KUKA KRL program: MyProgram_217().src

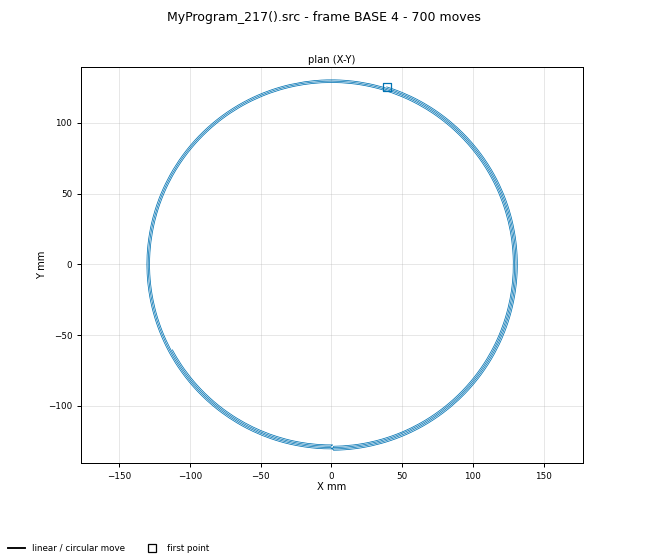
[picture p0: tool path of MyProgram_217().src in frame BASE 4, 700 of 700 moves have a stored position in this frame; points joined in program order, loops and branches not executed]
&ACCESS RVP
&REL 1
&PARAM TEMPLATE = C:\KRC\Roboter\Template\vorgabe
&PARAM EDITMASK = *
DEF MyProgram_217()
; ---- Setting reference (Base) ----
$BASE = BASE_DATA[4]

; --------------------------
; ---- Setting tool (TCP) ----
$TOOL = TOOL_DATA[3]
; --------------------------

$VEL.CP = VEL_APROX_PRINT
Startdeposition()
$VEL.CP = VEL_PRINT
LIN {X 39.0759,Y 125.4195,Z 152,A 69.1169,B 22.3843,C -1.1752,E1 22.4627,E2 378.1488} C_DIS
LIN {X 42.8509,Y 124.1788,Z 152,A 67.5035,B 22.3841,C -1.1792,E1 22.4669,E2 379.7481} C_DIS
LIN {X 46.0202,Y 123.0393,Z 152,A 66.1217,B 22.384,C -1.1819,E1 22.4705,E2 381.1197} C_DIS
LIN {X 49.9531,Y 121.4979,Z 152,A 64.0828,B 22.3845,C -1.1709,E1 22.4758,E2 383.1823} C_DIS
LIN {X 53.3923,Y 120.0244,Z 152,A 62.6413,B 22.3842,C -1.1779,E1 22.4795,E2 384.6014} C_DIS
LIN {X 55.8372,Y 118.9089,Z 152,A 61.2764,B 22.3847,C -1.1675,E1 22.483,E2 385.9896} C_DIS
LIN {X 59.0575,Y 117.3417,Z 152,A 59.7473,B 22.3847,C -1.167,E1 22.4868,E2 387.5152} C_DIS
LIN {X 62.6882,Y 115.4438,Z 152,A 57.9615,B 22.3848,C -1.1646,E1 22.4912,E2 389.3015} C_DIS
LIN {X 65.3716,Y 113.9459,Z 152,A 56.5252,B 22.3851,C -1.1582,E1 22.4947,E2 390.7497} C_DIS
LIN {X 69.7331,Y 111.3304,Z 152,A 54.6879,B 22.3844,C -1.1727,E1 22.499,E2 392.5428} C_DIS
LIN {X 72.7495,Y 109.3827,Z 152,A 52.8465,B 22.3852,C -1.1572,E1 22.5034,E2 394.4178} C_DIS
LIN {X 76.5216,Y 106.7777,Z 152,A 50.8731,B 22.3852,C -1.155,E1 22.5079,E2 396.3891} C_DIS
LIN {X 80.0679,Y 104.1454,Z 152,A 48.9647,B 22.3854,C -1.1524,E1 22.5121,E2 398.2966} C_DIS
LIN {X 83.4471,Y 101.4582,Z 152,A 47.0498,B 22.3857,C -1.1473,E1 22.5163,E2 400.2166} C_DIS
LIN {X 86.8041,Y 98.6009,Z 152,A 45.3735,B 22.3853,C -1.1552,E1 22.5198,E2 401.8648} C_DIS
LIN {X 88.621,Y 96.9709,Z 152,A 44.0641,B 22.3859,C -1.1415,E1 22.5226,E2 403.2042} C_DIS
LIN {X 92.4956,Y 93.2824,Z 152,A 41.7817,B 22.3861,C -1.1389,E1 22.5271,E2 405.4825} C_DIS
LIN {X 95.519,Y 90.1839,Z 152,A 39.8997,B 22.3862,C -1.1351,E1 22.5308,E2 407.3654} C_DIS
LIN {X 98.6375,Y 86.7627,Z 152,A 37.8778,B 22.3865,C -1.1304,E1 22.5346,E2 409.3894} C_DIS
LIN {X 101.415,Y 83.4994,Z 152,A 36.2489,B 22.3861,C -1.1374,E1 22.5374,E2 410.9914} C_DIS
LIN {X 103.0184,Y 81.5129,Z 152,A 34.8749,B 22.3869,C -1.1223,E1 22.5399,E2 412.3977} C_DIS
LIN {X 105.772,Y 77.9059,Z 152,A 32.9472,B 22.3869,C -1.1199,E1 22.5431,E2 414.3213} C_DIS
LIN {X 107.9986,Y 74.7891,Z 152,A 31.2247,B 22.3873,C -1.1132,E1 22.5459,E2 416.0518} C_DIS
LIN {X 110.566,Y 70.9379,Z 152,A 29.2946,B 22.3873,C -1.1122,E1 22.5488,E2 417.9735} C_DIS
LIN {X 112.9802,Y 67.0265,Z 152,A 27.2685,B 22.3876,C -1.1058,E1 22.5518,E2 420.0046} C_DIS
LIN {X 115.1352,Y 63.254,Z 152,A 25.4004,B 22.3878,C -1.102,E1 22.5543,E2 421.8718} C_DIS
LIN {X 116.9711,Y 59.7855,Z 152,A 23.8677,B 22.3876,C -1.1059,E1 22.5563,E2 423.385} C_DIS
LIN {X 118.8063,Y 56.0533,Z 152,A 21.862,B 22.3883,C -1.0915,E1 22.5587,E2 425.4161} C_DIS
LIN {X 120.4751,Y 52.3674,Z 152,A 20.2435,B 22.3883,C -1.0935,E1 22.5605,E2 427.0193} C_DIS
LIN {X 121.5852,Y 49.7396,Z 152,A 19.0427,B 22.3883,C -1.092,E1 22.5618,E2 428.2167} C_DIS
LIN {X 123.0594,Y 45.9666,Z 152,A 17.2165,B 22.3887,C -1.084,E1 22.5637,E2 430.0524} C_DIS
LIN {X 124.4991,Y 41.9132,Z 152,A 15.3852,B 22.3888,C -1.0805,E1 22.5653,E2 431.881} C_DIS
LIN {X 125.5845,Y 38.537,Z 152,A 13.7778,B 22.3892,C -1.0729,E1 22.5667,E2 433.4979} C_DIS
LIN {X 126.8539,Y 34.1282,Z 152,A 11.8493,B 22.3892,C -1.0704,E1 22.5681,E2 435.4206} C_DIS
LIN {X 127.5693,Y 31.3524,Z 152,A 10.4272,B 22.3898,C -1.0581,E1 22.5691,E2 436.8654} C_DIS
LIN {X 128.3238,Y 28.1021,Z 152,A 8.5123,B 22.391,C -1.0313,E1 22.5703,E2 438.8375} C_DIS
LIN {X 129.3311,Y 23.0236,Z 152,A 6.9093,B 22.3899,C -1.056,E1 22.5711,E2 440.3655} C_DIS
LIN {X 129.9659,Y 19.125,Z 152,A 5.1562,B 22.3902,C -1.0491,E1 22.5718,E2 442.1251} C_DIS
LIN {X 130.4075,Y 15.8299,Z 152,A 3.6744,B 22.3905,C -1.043,E1 22.5723,E2 443.613} C_DIS
LIN {X 130.9161,Y 10.8465,Z 152,A 1.5967,B 22.3905,C -1.0412,E1 22.5729,E2 445.6813} C_DIS
LIN {X 131.1931,Y 6.7104,Z 152,A -0.1239,B 22.3906,C -1.0397,E1 22.5732,E2 447.3943} C_DIS
LIN {X 131.3377,Y 2.7109,Z 152,A -1.9941,B 22.3912,C -1.028,E1 22.5733,E2 449.2825} C_DIS
LIN {X 131.3529,Y -1.7959,Z 152,A -3.9022,B 22.3913,C -1.0245,E1 22.5733,E2 451.187} C_DIS
LIN {X 131.2356,Y -5.864,Z 152,A -5.7352,B 22.3917,C -1.0159,E1 22.5731,E2 453.0299} C_DIS
LIN {X 131.0106,Y -9.6365,Z 152,A -7.2728,B 22.3917,C -1.0161,E1 22.5728,E2 454.5569} C_DIS
LIN {X 130.6589,Y -13.604,Z 152,A -9.1407,B 22.3922,C -1.004,E1 22.5723,E2 456.4436} C_DIS
LIN {X 130.0858,Y -18.286,Z 152,A -11.0585,B 22.3922,C -1.0043,E1 22.5716,E2 458.348} C_DIS
LIN {X 129.5248,Y -21.9092,Z 152,A -12.6685,B 22.3924,C -0.9986,E1 22.5709,E2 459.9622} C_DIS
LIN {X 128.7591,Y -26.0326,Z 152,A -14.5575,B 22.3928,C -0.9898,E1 22.5699,E2 461.8616} C_DIS
LIN {X 127.7964,Y -30.4103,Z 152,A -16.4042,B 22.3928,C -0.9889,E1 22.5687,E2 463.6986} C_DIS
LIN {X 126.9735,Y -33.6799,Z 152,A -17.7135,B 22.3927,C -0.9921,E1 22.5678,E2 464.9909} C_DIS
LIN {X 126.1061,Y -36.7942,Z 152,A -19.2732,B 22.3932,C -0.9804,E1 22.5666,E2 466.5712} C_DIS
LIN {X 124.8598,Y -40.8297,Z 152,A -21.1531,B 22.3935,C -0.9727,E1 22.565,E2 468.459} C_DIS
LIN {X 123.6518,Y -44.3489,Z 152,A -22.6966,B 22.3935,C -0.9716,E1 22.5636,E2 469.9957} C_DIS
LIN {X 122.4904,Y -47.462,Z 152,A -24.0809,B 22.3935,C -0.9703,E1 22.5622,E2 471.3746} C_DIS
LIN {X 120.3805,Y -52.5861,Z 152,A -26.6321,B 22.3942,C -0.9564,E1 22.5595,E2 473.9463} C_DIS
LIN {X 118.6274,Y -56.4278,Z 152,A -28.3416,B 22.3942,C -0.9573,E1 22.5575,E2 475.6429} C_DIS
LIN {X 115.2676,Y -63.0113,Z 152,A -31.5961,B 22.3946,C -0.9462,E1 22.5533,E2 478.9068} C_DIS
LIN {X 113.0629,Y -66.8877,Z 152,A -33.5919,B 22.3949,C -0.9381,E1 22.5504,E2 480.9122} C_DIS
LIN {X 110.7037,Y -70.7228,Z 152,A -35.4887,B 22.3949,C -0.9358,E1 22.5476,E2 482.8041} C_DIS
LIN {X 108.293,Y -74.3616,Z 152,A -37.3931,B 22.3952,C -0.9305,E1 22.5447,E2 484.7118} C_DIS
LIN {X 105.6688,Y -78.0464,Z 152,A -39.3055,B 22.3952,C -0.9281,E1 22.5415,E2 486.6201} C_DIS
LIN {X 103.8884,Y -80.4004,Z 152,A -40.7022,B 22.3956,C -0.9193,E1 22.5391,E2 488.0322} C_DIS
LIN {X 101.1979,Y -83.7616,Z 152,A -43.1794,B 22.3969,C -0.8855,E1 22.5346,E2 490.5846} C_DIS
LIN {X 97.4652,Y -88.0773,Z 152,A -45.38,B 22.3966,C -0.893,E1 22.5306,E2 492.7545} C_DIS
LIN {X 94.5654,Y -91.183,Z 152,A -46.9074,B 22.3962,C -0.9041,E1 22.5277,E2 494.2455} C_DIS
LIN {X 89.8695,Y -95.8156,Z 152,A -49.6238,B 22.3962,C -0.905,E1 22.5223,E2 496.9468} C_DIS
LIN {X 84.2334,Y -100.8059,Z 152,A -52.7429,B 22.3962,C -0.9054,E1 22.5158,E2 500.0509} C_DIS
LIN {X 82.4164,Y -102.2964,Z 152,A -54.3606,B 22.3973,C -0.8747,E1 22.5121,E2 501.7419} C_DIS
LIN {X 79.0783,Y -104.8983,Z 152,A -56.1035,B 22.3973,C -0.8758,E1 22.5082,E2 503.475} C_DIS
LIN {X 76.025,Y -107.1324,Z 152,A -57.4826,B 22.3969,C -0.8853,E1 22.5051,E2 504.8237} C_DIS
LIN {X 72.219,Y -109.7335,Z 152,A -59.4323,B 22.3969,C -0.8843,E1 22.5006,E2 506.7687} C_DIS
LIN {X 68.385,Y -112.1635,Z 152,A -61.4412,B 22.3972,C -0.8792,E1 22.4958,E2 508.7837} C_DIS
LIN {X 64.5104,Y -114.4354,Z 152,A -63.3541,B 22.3972,C -0.8779,E1 22.4912,E2 510.6936} C_DIS
LIN {X 60.7291,Y -116.4844,Z 152,A -65.095,B 22.3971,C -0.8811,E1 22.487,E2 512.4203} C_DIS
LIN {X 56.5099,Y -118.5882,Z 152,A -67.198,B 22.3973,C -0.8756,E1 22.4817,E2 514.5314} C_DIS
LIN {X 53.0564,Y -120.1746,Z 152,A -68.9498,B 22.3976,C -0.8686,E1 22.4772,E2 516.2966} C_DIS
LIN {X 49.5085,Y -121.6783,Z 152,A -70.4769,B 22.3974,C -0.8735,E1 22.4733,E2 517.807} C_DIS
LIN {X 45.1537,Y -123.3616,Z 152,A -72.6362,B 22.3977,C -0.8649,E1 22.4676,E2 519.9834} C_DIS
LIN {X 41.6015,Y -124.6029,Z 152,A -74.081,B 22.3974,C -0.8722,E1 22.4639,E2 521.406} C_DIS
LIN {X 38.537,Y -125.5845,Z 152,A -75.5338,B 22.3976,C -0.8682,E1 22.46,E2 522.8662} C_DIS
LIN {X 35.354,Y -126.5174,Z 152,A -76.8689,B 22.3974,C -0.8719,E1 22.4564,E2 524.1891} C_DIS
LIN {X 31.0295,Y -127.6472,Z 152,A -78.8275,B 22.3975,C -0.8694,E1 22.4511,E2 526.1506} C_DIS
LIN {X 28.7199,Y -128.1875,Z 152,A -80.4521,B 22.3986,C -0.841,E1 22.4465,E2 527.8474} C_DIS
LIN {X 24.8562,Y -128.9914,Z 152,A -82.107,B 22.3985,C -0.8426,E1 22.442,E2 529.4957} C_DIS
LIN {X 21.1843,Y -129.6457,Z 152,A -83.4884,B 22.3981,C -0.8528,E1 22.4382,E2 530.8489} C_DIS
LIN {X 16.9785,Y -130.2626,Z 152,A -85.2127,B 22.398,C -0.8576,E1 22.4335,E2 532.5589} C_DIS
LIN {X 12.8893,Y -130.731,Z 152,A -87.043,B 22.398,C -0.855,E1 22.4284,E2 534.3946} C_DIS
LIN {X 9.8072,Y -130.9981,Z 152,A -88.5323,B 22.3983,C -0.8479,E1 22.4242,E2 535.9016} C_DIS
LIN {X 5.3117,Y -131.2573,Z 152,A -90.3189,B 22.398,C -0.8553,E1 22.4193,E2 537.668} C_DIS
LIN {X 1.4511,Y -131.3586,Z 152,A -92.1085,B 22.3982,C -0.85,E1 22.4143,E2 539.4713} C_DIS
LIN {X 1.4511,Y -131.3586,Z 152,A -92.1085,B 22.3982,C -0.85,E1 22.4143,E2 539.4713} C_DIS
Enddeposition()
LIN {X 0.9252,Y -130.4174,Z 152,A -91.4009,B 21.3974,C -0.7347,E1 21.4116,E2 538.9603} C_DIS
Startdeposition()
$VEL.CP = VEL_PRINT
LIN {X 4.401,Y -130.3502,Z 152,A -89.5833,B 21.397,C -0.7479,E1 21.4168,E2 537.1069} C_DIS
LIN {X 7.5621,Y -130.2041,Z 152,A -87.7196,B 21.3963,C -0.7696,E1 21.4221,E2 535.1847} C_DIS
LIN {X 12.3533,Y -129.8363,Z 152,A -86.2062,B 21.3971,C -0.7439,E1 21.4261,E2 533.7428} C_DIS
LIN {X 16.3199,Y -129.399,Z 152,A -84.4088,B 21.3971,C -0.7469,E1 21.4311,E2 531.9389} C_DIS
LIN {X 22.9385,Y -128.3895,Z 152,A -81.4914,B 21.3971,C -0.7479,E1 21.4392,E2 529.0222} C_DIS
LIN {X 29.5447,Y -127.033,Z 152,A -78.4786,B 21.3968,C -0.7527,E1 21.4474,E2 526.0009} C_DIS
LIN {X 34.0528,Y -125.8993,Z 152,A -76.4296,B 21.3968,C -0.755,E1 21.453,E2 523.9493} C_DIS
LIN {X 38.0089,Y -124.7611,Z 152,A -74.7239,B 21.3968,C -0.7524,E1 21.4575,E2 522.2544} C_DIS
LIN {X 41.3367,Y -123.6984,Z 152,A -73.2639,B 21.3969,C -0.7508,E1 21.4614,E2 520.8018} C_DIS
LIN {X 44.246,Y -122.6877,Z 152,A -71.909,B 21.3969,C -0.7526,E1 21.4649,E2 519.4454} C_DIS
LIN {X 51.5801,Y -119.7894,Z 152,A -68.4066,B 21.3966,C -0.759,E1 21.474,E2 515.9348} C_DIS
LIN {X 54.631,Y -118.429,Z 152,A -66.0213,B 21.3951,C -0.8034,E1 21.4804,E2 513.4355} C_DIS
LIN {X 60.4214,Y -115.5822,Z 152,A -64.14,B 21.3965,C -0.7641,E1 21.4848,E2 511.6678} C_DIS
LIN {X 64.2221,Y -113.517,Z 152,A -62.1023,B 21.3961,C -0.7736,E1 21.4898,E2 509.6112} C_DIS
LIN {X 68.0638,Y -111.2555,Z 152,A -60.1772,B 21.3961,C -0.7757,E1 21.4944,E2 507.6876} C_DIS
LIN {X 71.6684,Y -108.9683,Z 152,A -58.3196,B 21.396,C -0.7784,E1 21.4987,E2 505.8297} C_DIS
LIN {X 75.4742,Y -106.3684,Z 152,A -56.4222,B 21.396,C -0.7766,E1 21.503,E2 503.9451} C_DIS
LIN {X 77.6887,Y -104.7616,Z 152,A -55.2144,B 21.396,C -0.7793,E1 21.5058,E2 502.735} C_DIS
LIN {X 82.2112,Y -101.2519,Z 152,A -52.5747,B 21.3955,C -0.7904,E1 21.5116,E2 500.0766} C_DIS
LIN {X 85.2765,Y -98.6834,Z 152,A -50.4735,B 21.3948,C -0.8103,E1 21.5161,E2 497.9308} C_DIS
LIN {X 88.3815,Y -95.9124,Z 152,A -48.5103,B 21.3945,C -0.8209,E1 21.5202,E2 495.9483} C_DIS
LIN {X 91.9267,Y -92.5199,Z 152,A -46.9023,B 21.3952,C -0.8004,E1 21.5233,E2 494.4042} C_DIS
LIN {X 97.2688,Y -86.8865,Z 152,A -43.0456,B 21.3941,C -0.8297,E1 21.5307,E2 490.4879} C_DIS
LIN {X 100.2547,Y -83.4239,Z 152,A -41.4961,B 21.3947,C -0.8133,E1 21.5334,E2 488.9914} C_DIS
LIN {X 102.7993,Y -80.2677,Z 152,A -39.7139,B 21.3946,C -0.818,E1 21.5365,E2 487.2063} C_DIS
LIN {X 105.4275,Y -76.7827,Z 152,A -37.8044,B 21.3944,C -0.8228,E1 21.5396,E2 485.2947} C_DIS
LIN {X 107.8695,Y -73.3123,Z 152,A -35.9707,B 21.3942,C -0.8265,E1 21.5426,E2 483.4617} C_DIS
LIN {X 110.366,Y -69.4969,Z 152,A -34.0103,B 21.3942,C -0.8301,E1 21.5455,E2 481.5032} C_DIS
LIN {X 112.6618,Y -65.711,Z 152,A -32.0287,B 21.3938,C -0.8373,E1 21.5483,E2 479.5141} C_DIS
LIN {X 114.6698,Y -62.1403,Z 152,A -29.1425,B 21.3917,C -0.8941,E1 21.5524,E2 476.4911} C_DIS
LIN {X 118.2409,Y -55.0378,Z 152,A -26.9035,B 21.3936,C -0.8448,E1 21.5549,E2 474.4006} C_DIS
LIN {X 121.0471,Y -48.5553,Z 152,A -23.7639,B 21.3931,C -0.8559,E1 21.5583,E2 471.2514} C_DIS
LIN {X 122.9923,Y -43.398,Z 152,A -21.3202,B 21.3928,C -0.8643,E1 21.5607,E2 468.801} C_DIS
LIN {X 124.1626,Y -39.921,Z 152,A -19.8445,B 21.3928,C -0.8629,E1 21.5619,E2 467.339} C_DIS
LIN {X 125.0716,Y -36.9756,Z 152,A -18.4548,B 21.3926,C -0.8688,E1 21.563,E2 465.9428} C_DIS
LIN {X 125.9647,Y -33.8073,Z 152,A -17.0128,B 21.3925,C -0.8731,E1 21.5641,E2 464.4988} C_DIS
LIN {X 126.9017,Y -30.1032,Z 152,A -15.3229,B 21.3923,C -0.8789,E1 21.5652,E2 462.8047} C_DIS
LIN {X 127.7436,Y -26.3,Z 152,A -13.6339,B 21.3921,C -0.8832,E1 21.5662,E2 461.1156} C_DIS
LIN {X 128.6323,Y -21.5356,Z 152,A -11.5618,B 21.3919,C -0.8873,E1 21.5672,E2 459.0468} C_DIS
LIN {X 129.1811,Y -17.9597,Z 152,A -10.0533,B 21.3919,C -0.8885,E1 21.5678,E2 457.5455} C_DIS
LIN {X 129.7907,Y -12.8285,Z 152,A -7.6059,B 21.3913,C -0.9041,E1 21.5686,E2 455.0729} C_DIS
LIN {X 130.1561,Y -8.3413,Z 152,A -5.7478,B 21.3913,C -0.9048,E1 21.569,E2 453.226} C_DIS
LIN {X 130.3399,Y -4.6658,Z 152,A -4.06,B 21.3909,C -0.9133,E1 21.5692,E2 451.527} C_DIS
LIN {X 130.4182,Y 1.2459,Z 152,A -1.5813,B 21.3908,C -0.916,E1 21.5692,E2 449.0586} C_DIS
LIN {X 130.2441,Y 6.8284,Z 152,A 0.9539,B 21.3903,C -0.9276,E1 21.569,E2 446.5096} C_DIS
LIN {X 129.9978,Y 10.5288,Z 152,A 2.8599,B 21.3895,C -0.9458,E1 21.5685,E2 444.5673} C_DIS
LIN {X 129.6462,Y 14.2119,Z 152,A 4.8108,B 21.3887,C -0.9664,E1 21.5679,E2 442.5741} C_DIS
LIN {X 128.9348,Y 19.646,Z 152,A 6.4917,B 21.3898,C -0.9396,E1 21.5673,E2 440.9781} C_DIS
LIN {X 128.1808,Y 24.0808,Z 152,A 8.89,B 21.3887,C -0.9656,E1 21.566,E2 438.5257} C_DIS
LIN {X 127.3556,Y 28.1238,Z 152,A 10.306,B 21.3893,C -0.9524,E1 21.5652,E2 437.1552} C_DIS
LIN {X 126.4429,Y 31.9722,Z 152,A 12.0043,B 21.3891,C -0.9559,E1 21.5641,E2 435.4592} C_DIS
LIN {X 125.3275,Y 36.1016,Z 152,A 13.8644,B 21.3889,C -0.9607,E1 21.5627,E2 433.5987} C_DIS
LIN {X 124.2876,Y 39.5299,Z 152,A 15.3719,B 21.3889,C -0.9623,E1 21.5614,E2 432.097} C_DIS
LIN {X 123.2775,Y 42.5754,Z 152,A 16.646,B 21.3889,C -0.9602,E1 21.5603,E2 430.8372} C_DIS
LIN {X 122.252,Y 45.4371,Z 152,A 17.902,B 21.3889,C -0.9604,E1 21.5591,E2 429.589} C_DIS
LIN {X 120.3818,Y 50.1816,Z 152,A 20.3347,B 21.3882,C -0.9758,E1 21.5566,E2 427.1303} C_DIS
LIN {X 119.1157,Y 53.117,Z 152,A 21.7307,B 21.3881,C -0.9794,E1 21.555,E2 425.7336} C_DIS
LIN {X 116.6426,Y 58.3522,Z 152,A 24.2935,B 21.3877,C -0.9874,E1 21.5519,E2 423.1655} C_DIS
LIN {X 114.6934,Y 62.0971,Z 152,A 26.1776,B 21.3875,C -0.9938,E1 21.5494,E2 421.2756} C_DIS
LIN {X 112.7049,Y 65.6367,Z 152,A 28.1741,B 21.3868,C -1.0085,E1 21.5466,E2 419.2513} C_DIS
LIN {X 111.0193,Y 68.449,Z 152,A 29.4001,B 21.3871,C -1.0023,E1 21.5448,E2 418.0497} C_DIS
LIN {X 109.0601,Y 71.529,Z 152,A 31.3509,B 21.3862,C -1.0225,E1 21.5418,E2 416.0552} C_DIS
LIN {X 106.7687,Y 74.9067,Z 152,A 32.7995,B 21.3867,C -1.0111,E1 21.5396,E2 414.6463} C_DIS
LIN {X 104.2205,Y 78.4128,Z 152,A 34.5911,B 21.3867,C -1.0106,E1 21.5366,E2 412.8664} C_DIS
LIN {X 102.4656,Y 80.6925,Z 152,A 35.9867,B 21.3863,C -1.0197,E1 21.5342,E2 411.4537} C_DIS
LIN {X 99.4954,Y 84.3277,Z 152,A 37.9726,B 21.3863,C -1.021,E1 21.5306,E2 409.4752} C_DIS
LIN {X 96.5683,Y 87.6642,Z 152,A 39.8898,B 21.3861,C -1.0239,E1 21.5271,E2 407.5601} C_DIS
LIN {X 93.5342,Y 90.8948,Z 152,A 41.8395,B 21.3859,C -1.0283,E1 21.5233,E2 405.6085} C_DIS
LIN {X 90.9016,Y 93.5276,Z 152,A 43.2146,B 21.3863,C -1.0198,E1 21.5206,E2 404.2633} C_DIS
LIN {X 87.7999,Y 96.4452,Z 152,A 45.3159,B 21.3856,C -1.0342,E1 21.5163,E2 402.1331} C_DIS
LIN {X 84.5912,Y 99.2714,Z 152,A 47.1871,B 21.3855,C -1.0375,E1 21.5123,E2 400.2614} C_DIS
LIN {X 81.2269,Y 102.0423,Z 152,A 49.103,B 21.3853,C -1.0412,E1 21.5082,E2 398.3443} C_DIS
LIN {X 77.5965,Y 104.8302,Z 152,A 51.1325,B 21.3851,C -1.0456,E1 21.5036,E2 396.3114} C_DIS
LIN {X 74.0641,Y 107.3549,Z 152,A 52.8328,B 21.3854,C -1.0395,E1 21.4998,E2 394.6348} C_DIS
LIN {X 70.5474,Y 109.6977,Z 152,A 54.8702,B 21.3849,C -1.0506,E1 21.495,E2 392.5749} C_DIS
LIN {X 67.7525,Y 111.4457,Z 152,A 56.7306,B 21.3839,C -1.0714,E1 21.4904,E2 390.6647} C_DIS
LIN {X 63.9819,Y 113.652,Z 152,A 58.2119,B 21.3847,C -1.0544,E1 21.487,E2 389.235} C_DIS
LIN {X 59.9161,Y 115.8476,Z 152,A 60.2401,B 21.3846,C -1.057,E1 21.4819,E2 387.2064} C_DIS
LIN {X 56.4723,Y 117.5623,Z 152,A 62.0593,B 21.3842,C -1.065,E1 21.4773,E2 385.3713} C_DIS
LIN {X 52.0411,Y 119.59,Z 152,A 63.9461,B 21.3846,C -1.0561,E1 21.4726,E2 383.5143} C_DIS
LIN {X 45.5953,Y 122.1927,Z 152,A 67.0474,B 21.3844,C -1.0613,E1 21.4645,E2 380.4071} C_DIS
LIN {X 41.5578,Y 123.6247,Z 152,A 68.8825,B 21.3844,C -1.0609,E1 21.4597,E2 378.5775} C_DIS
LIN {X 38.2417,Y 124.6899,Z 152,A 70.417,B 21.3844,C -1.0623,E1 21.4556,E2 377.0424} C_DIS
LIN {X 35.3722,Y 125.5344,Z 152,A 71.6767,B 21.3844,C -1.0608,E1 21.4523,E2 375.7893} C_DIS
LIN {X 32.5433,Y 126.2979,Z 152,A 72.9777,B 21.3844,C -1.0623,E1 21.4487,E2 374.4868} C_DIS
LIN {X 29.9299,Y 126.9434,Z 152,A 74.1576,B 21.3843,C -1.0628,E1 21.4455,E2 373.3073} C_DIS
LIN {X 26.5227,Y 127.6983,Z 152,A 75.5949,B 21.3845,C -1.0595,E1 21.4416,E2 371.8815} C_DIS
LIN {X 22.6421,Y 128.4425,Z 152,A 77.5846,B 21.3839,C -1.0713,E1 21.4361,E2 369.8621} C_DIS
LIN {X 19.7595,Y 128.9172,Z 152,A 79.2572,B 21.3831,C -1.0887,E1 21.4314,E2 368.1436} C_DIS
LIN {X 15.4579,Y 129.5033,Z 152,A 80.906,B 21.3836,C -1.0778,E1 21.4269,E2 366.5261} C_DIS
LIN {X 10.141,Y 130.0294,Z 152,A 83.0703,B 21.3839,C -1.0701,E1 21.4209,E2 364.3844} C_DIS
LIN {X 6.1136,Y 130.2801,Z 152,A 85.1972,B 21.3832,C -1.0855,E1 21.4149,E2 362.2162} C_DIS
LIN {X 2.2497,Y 130.4034,Z 152,A 86.4789,B 21.3841,C -1.0673,E1 21.4114,E2 360.9846} C_DIS
LIN {X -3.3097,Y 130.3811,Z 152,A 88.9249,B 21.3841,C -1.067,E1 21.4046,E2 358.5395} C_DIS
LIN {X -7.1528,Y 130.2278,Z 152,A 90.5486,B 21.3843,C -1.0636,E1 21.4001,E2 356.9245} C_DIS
LIN {X -12.0515,Y 129.8653,Z 152,A 92.889,B 21.3839,C -1.0705,E1 21.3935,E2 354.564} C_DIS
LIN {X -19.2417,Y 128.9974,Z 152,A 95.9908,B 21.3842,C -1.0653,E1 21.385,E2 351.4739} C_DIS
LIN {X -29.4048,Y 127.065,Z 152,A 100.5028,B 21.3844,C -1.0602,E1 21.3727,E2 346.9697} C_DIS
LIN {X -32.8429,Y 126.2219,Z 152,A 102.1955,B 21.3842,C -1.0646,E1 21.368,E2 345.2623} C_DIS
LIN {X -36.4995,Y 125.211,Z 152,A 103.675,B 21.3847,C -1.055,E1 21.3641,E2 343.8062} C_DIS
LIN {X -39.5106,Y 124.2938,Z 152,A 105.1,B 21.3847,C -1.0553,E1 21.3603,E2 342.3776} C_DIS
LIN {X -42.6828,Y 123.2403,Z 152,A 106.5262,B 21.3848,C -1.0518,E1 21.3565,E2 340.9577} C_DIS
LIN {X -48.1229,Y 121.2214,Z 152,A 109.0803,B 21.385,C -1.0487,E1 21.3499,E2 338.4059} C_DIS
LIN {X -51.8586,Y 119.6689,Z 152,A 111.3754,B 21.3841,C -1.0679,E1 21.3438,E2 336.0517} C_DIS
LIN {X -55.5846,Y 117.9864,Z 152,A 112.8302,B 21.3849,C -1.0509,E1 21.3403,E2 334.6392} C_DIS
LIN {X -58.7992,Y 116.4164,Z 152,A 114.3679,B 21.385,C -1.0471,E1 21.3364,E2 333.1072} C_DIS
LIN {X -62,Y 114.7456,Z 152,A 116.0094,B 21.385,C -1.0467,E1 21.3324,E2 331.4613} C_DIS
LIN {X -65.797,Y 112.6113,Z 152,A 117.9466,B 21.3852,C -1.0444,E1 21.3277,E2 329.5236} C_DIS
LIN {X -69.6155,Y 110.2911,Z 152,A 120.4492,B 21.3843,C -1.0632,E1 21.3216,E2 326.9597} C_DIS
LIN {X -73.809,Y 107.5299,Z 152,A 122.0851,B 21.3856,C -1.0354,E1 21.318,E2 325.3941} C_DIS
LIN {X -77.3446,Y 105.0156,Z 152,A 124.0057,B 21.3857,C -1.0322,E1 21.3136,E2 323.4742} C_DIS
LIN {X -80.8493,Y 102.3425,Z 152,A 125.9441,B 21.3859,C -1.0282,E1 21.3094,E2 321.5383} C_DIS
LIN {X -84.1132,Y 99.6773,Z 152,A 127.8475,B 21.3859,C -1.0264,E1 21.3053,E2 319.6313} C_DIS
LIN {X -87.3861,Y 96.8206,Z 152,A 129.7851,B 21.3861,C -1.0233,E1 21.3012,E2 317.6931} C_DIS
LIN {X -90.7047,Y 93.7182,Z 152,A 131.7135,B 21.3865,C -1.0159,E1 21.2974,E2 315.7756} C_DIS
LIN {X -93.6474,Y 90.7779,Z 152,A 133.5847,B 21.3865,C -1.0134,E1 21.2937,E2 313.9019} C_DIS
LIN {X -96.7679,Y 87.4442,Z 152,A 135.6037,B 21.3868,C -1.009,E1 21.2899,E2 311.8845} C_DIS
LIN {X -99.656,Y 84.1386,Z 152,A 137.5847,B 21.3869,C -1.0062,E1 21.2863,E2 309.9002} C_DIS
LIN {X -102.5063,Y 80.6407,Z 152,A 139.5472,B 21.3872,C -1.0003,E1 21.2828,E2 307.9432} C_DIS
LIN {X -105.293,Y 76.9671,Z 152,A 141.5964,B 21.3874,C -0.9959,E1 21.2794,E2 305.8944} C_DIS
LIN {X -107.8201,Y 73.3852,Z 152,A 143.4904,B 21.3877,C -0.9894,E1 21.2764,E2 304.0072} C_DIS
LIN {X -111.8691,Y 67.0512,Z 152,A 146.8797,B 21.3879,C -0.9836,E1 21.2714,E2 300.6132} C_DIS
LIN {X -114.0485,Y 63.2725,Z 152,A 148.7078,B 21.3883,C -0.9746,E1 21.2689,E2 298.7986} C_DIS
LIN {X -117.2922,Y 57.0355,Z 152,A 151.8936,B 21.3885,C -0.9695,E1 21.2649,E2 295.6066} C_DIS
LIN {X -118.8109,Y 53.7985,Z 152,A 153.3731,B 21.3889,C -0.9612,E1 21.2631,E2 294.1403} C_DIS
LIN {X -120.5023,Y 49.8932,Z 152,A 155.4256,B 21.3889,C -0.963,E1 21.2609,E2 292.0695} C_DIS
LIN {X -121.735,Y 46.806,Z 152,A 156.9784,B 21.3889,C -0.9622,E1 21.2593,E2 290.5083} C_DIS
LIN {X -123.468,Y 42.0258,Z 152,A 159.1147,B 21.3893,C -0.9515,E1 21.2574,E2 288.3873} C_DIS
LIN {X -124.5452,Y 38.7144,Z 152,A 161.3689,B 21.3882,C -0.976,E1 21.2555,E2 286.0499} C_DIS
LIN {X -126.1925,Y 32.9532,Z 152,A 163.3261,B 21.3898,C -0.9405,E1 21.2541,E2 284.1773} C_DIS
LIN {X -127.1359,Y 29.0945,Z 152,A 164.9195,B 21.3902,C -0.929,E1 21.2531,E2 282.6045} C_DIS
LIN {X -127.8318,Y 25.8665,Z 152,A 166.4129,B 21.3904,C -0.9261,E1 21.2522,E2 281.1085} C_DIS
LIN {X -128.5399,Y 22.0894,Z 152,A 168.1843,B 21.3904,C -0.9241,E1 21.2513,E2 279.3302} C_DIS
LIN {X -129.1696,Y 18.0397,Z 152,A 169.9747,B 21.3907,C -0.918,E1 21.2506,E2 277.544} C_DIS
LIN {X -129.7116,Y 13.6046,Z 152,A 172.2209,B 21.3905,C -0.9231,E1 21.2499,E2 275.2676} C_DIS
LIN {X -130.0279,Y 10.162,Z 152,A 173.8206,B 21.3905,C -0.9215,E1 21.2496,E2 273.6609} C_DIS
LIN {X -130.2565,Y 6.5831,Z 152,A 174.8744,B 21.3916,C -0.8956,E1 21.2494,E2 272.6711} C_DIS
LIN {X -130.4256,Y -0.1033,Z 152,A 177.9488,B 21.3918,C -0.8916,E1 21.2493,E2 269.5857} C_DIS
LIN {X -130.2528,Y -6.6552,Z 152,A -179.129,B 21.392,C -0.8842,E1 21.2495,E2 266.663} C_DIS
LIN {X -130.0182,Y -10.2864,Z 152,A -177.0912,B 21.3915,C -0.8967,E1 21.25,E2 264.5759} C_DIS
LIN {X -129.6719,Y -13.9728,Z 152,A -175.584,B 21.3919,C -0.8868,E1 21.2504,E2 263.0853} C_DIS
LIN {X -129.0069,Y -19.1783,Z 152,A -173.4227,B 21.3925,C -0.8738,E1 21.2512,E2 260.9446} C_DIS
LIN {X -128.4009,Y -22.8746,Z 152,A -171.8983,B 21.3928,C -0.8638,E1 21.2519,E2 259.4369} C_DIS
LIN {X -127.754,Y -26.2486,Z 152,A -170.3329,B 21.3929,C -0.8614,E1 21.2528,E2 257.8672} C_DIS
LIN {X -126.8384,Y -30.3656,Z 152,A -168.4934,B 21.3932,C -0.8552,E1 21.2539,E2 256.0319} C_DIS
LIN {X -126.0192,Y -33.6029,Z 152,A -166.9849,B 21.3932,C -0.8525,E1 21.255,E2 254.5206} C_DIS
LIN {X -124.8276,Y -37.7919,Z 152,A -165.1142,B 21.3936,C -0.845,E1 21.2565,E2 252.6576} C_DIS
LIN {X -123.8678,Y -40.8278,Z 152,A -163.3552,B 21.3932,C -0.8554,E1 21.258,E2 250.8579} C_DIS
LIN {X -122.773,Y -44.0092,Z 152,A -161.7971,B 21.3932,C -0.8544,E1 21.2595,E2 249.2922} C_DIS
LIN {X -121.4562,Y -47.523,Z 152,A -160.4671,B 21.3939,C -0.8366,E1 21.2608,E2 248.0023} C_DIS
LIN {X -119.895,Y -51.3357,Z 152,A -158.8673,B 21.3944,C -0.8229,E1 21.2625,E2 246.4297} C_DIS
LIN {X -118.4729,Y -54.536,Z 152,A -157.2039,B 21.3944,C -0.8236,E1 21.2644,E2 244.7534} C_DIS
LIN {X -117.0635,Y -57.499,Z 152,A -155.7156,B 21.3944,C -0.8215,E1 21.2662,E2 243.2614} C_DIS
LIN {X -115.2287,Y -61.0947,Z 152,A -153.6471,B 21.3942,C -0.8287,E1 21.269,E2 241.16} C_DIS
LIN {X -113.6926,Y -63.9093,Z 152,A -152.1678,B 21.3942,C -0.8278,E1 21.271,E2 239.6739} C_DIS
LIN {X -111.9486,Y -66.9179,Z 152,A -150.954,B 21.3948,C -0.8109,E1 21.2727,E2 238.4992} C_DIS
LIN {X -110.3728,Y -69.4861,Z 152,A -149.7103,B 21.3951,C -0.8042,E1 21.2745,E2 237.2664} C_DIS
LIN {X -108.4247,Y -72.4882,Z 152,A -147.9625,B 21.3949,C -0.8074,E1 21.2772,E2 235.4995} C_DIS
LIN {X -105.9036,Y -76.1248,Z 152,A -145.9907,B 21.3951,C -0.8037,E1 21.2804,E2 233.5263} C_DIS
LIN {X -103.2728,Y -79.6573,Z 152,A -144.0334,B 21.3952,C -0.7999,E1 21.2837,E2 231.5683} C_DIS
LIN {X -100.4336,Y -83.2079,Z 152,A -142.0663,B 21.3954,C -0.794,E1 21.2871,E2 229.6066} C_DIS
LIN {X -97.585,Y -86.5313,Z 152,A -140.0818,B 21.3954,C -0.7922,E1 21.2908,E2 227.6165} C_DIS
LIN {X -94.5093,Y -89.8808,Z 152,A -138.1171,B 21.3957,C -0.7864,E1 21.2945,E2 225.6574} C_DIS
LIN {X -91.692,Y -92.7531,Z 152,A -136.6058,B 21.3962,C -0.7721,E1 21.2975,E2 224.1781} C_DIS
LIN {X -87.8257,Y -96.4218,Z 152,A -133.9622,B 21.3959,C -0.7798,E1 21.3029,E2 221.5002} C_DIS
LIN {X -84.3224,Y -99.4998,Z 152,A -131.9342,B 21.3961,C -0.775,E1 21.3072,E2 219.476} C_DIS
LIN {X -80.9034,Y -102.2999,Z 152,A -129.9378,B 21.3961,C -0.7737,E1 21.3115,E2 217.4743} C_DIS
LIN {X -77.5355,Y -104.8754,Z 152,A -128.2211,B 21.3964,C -0.7644,E1 21.3153,E2 215.7761} C_DIS
LIN {X -72.5554,Y -108.3799,Z 152,A -125.5022,B 21.3965,C -0.7617,E1 21.3216,E2 213.0534} C_DIS
LIN {X -66.7585,Y -112.0436,Z 152,A -122.4004,B 21.3965,C -0.7609,E1 21.329,E2 209.9423} C_DIS
LIN {X -63.1574,Y -114.1122,Z 152,A -120.5831,B 21.3967,C -0.7581,E1 21.3334,E2 208.1265} C_DIS
LIN {X -59.8444,Y -115.8843,Z 152,A -119.0388,B 21.3969,C -0.7514,E1 21.3372,E2 206.5954} C_DIS
LIN {X -55.5587,Y -117.9988,Z 152,A -116.7773,B 21.3967,C -0.7558,E1 21.3429,E2 204.315} C_DIS
LIN {X -48.7648,Y -120.9626,Z 152,A -113.6584,B 21.397,C -0.7464,E1 21.3509,E2 201.2132} C_DIS
LIN {X -45.9016,Y -122.078,Z 152,A -112.3067,B 21.397,C -0.7452,E1 21.3544,E2 199.8614} C_DIS
LIN {X -42.878,Y -123.1726,Z 152,A -110.8508,B 21.397,C -0.7458,E1 21.3582,E2 198.4005} C_DIS
LIN {X -39.703,Y -124.2323,Z 152,A -109.4427,B 21.3972,C -0.742,E1 21.3619,E2 196.9998} C_DIS
LIN {X -36.334,Y -125.2595,Z 152,A -107.7466,B 21.397,C -0.7473,E1 21.3665,E2 195.2859} C_DIS
LIN {X -33.0699,Y -126.1614,Z 152,A -106.36,B 21.3972,C -0.742,E1 21.3702,E2 193.9114} C_DIS
LIN {X -29.3617,Y -127.0748,Z 152,A -104.6056,B 21.3972,C -0.7444,E1 21.375,E2 192.1475} C_DIS
LIN {X -25.0719,Y -127.9913,Z 152,A -102.6628,B 21.3972,C -0.7442,E1 21.3804,E2 190.2026} C_DIS
LIN {X -19.0198,Y -129.0296,Z 152,A -99.8408,B 21.397,C -0.7488,E1 21.3882,E2 187.3649} C_DIS
LIN {X -14.1339,Y -129.6546,Z 152,A -97.866,B 21.3973,C -0.7402,E1 21.3936,E2 185.4122} C_DIS
LIN {X -10.3274,Y -130.0148,Z 152,A -96.1744,B 21.3973,C -0.7405,E1 21.3983,E2 183.7187} C_DIS
LIN {X -5.3795,Y -130.3121,Z 152,A -94.003,B 21.3973,C -0.7403,E1 21.4044,E2 181.5471} C_DIS
LIN {X -1.6972,Y -130.4126,Z 152,A -92.2924,B 21.3971,C -0.7446,E1 21.4092,E2 179.8246} C_DIS
LIN {X 0.9252,Y -130.4174,Z 152,A -91.3977,B 21.3975,C -0.7336,E1 21.4116,E2 178.9603} C_DIS
Enddeposition()
LIN {X 0.9252,Y -130.4174,Z 152,A -91.3977,B 21.3975,C -0.7336,E1 21.4116,E2 178.9603} C_DIS
Startdeposition()
$VEL.CP = VEL_PRINT
LIN {X -0.5193,Y -129.4801,Z 152,A -92.2024,B 20.2005,C -0.5505,E1 20.2064,E2 180.1544} C_DIS
LIN {X -4.0171,Y -129.4193,Z 152,A -93.9054,B 20.2006,C -0.5441,E1 20.2016,E2 181.8763} C_DIS
LIN {X -9.319,Y -129.1451,Z 152,A -96.1087,B 20.2005,C -0.55,E1 20.1955,E2 184.0633} C_DIS
LIN {X -13.1881,Y -128.8091,Z 152,A -98.0602,B 20.2007,C -0.5407,E1 20.19,E2 186.0429} C_DIS
LIN {X -17.7326,Y -128.2621,Z 152,A -100.592,B 20.2012,C -0.521,E1 20.1828,E2 188.6343} C_DIS
LIN {X -23.0906,Y -127.4055,Z 152,A -102.8433,B 20.201,C -0.5278,E1 20.1767,E2 190.8688} C_DIS
LIN {X -27.7259,Y -126.478,Z 152,A -104.3802,B 20.2005,C -0.5509,E1 20.1727,E2 192.3412} C_DIS
LIN {X -32.1357,Y -125.4297,Z 152,A -106.3661,B 20.2005,C -0.5528,E1 20.1673,E2 194.3249} C_DIS
LIN {X -36.3677,Y -124.2683,Z 152,A -108.2798,B 20.2003,C -0.5552,E1 20.1621,E2 196.2355} C_DIS
LIN {X -39.4081,Y -123.3378,Z 152,A -109.7063,B 20.2003,C -0.5555,E1 20.1583,E2 197.6643} C_DIS
LIN {X -42.544,Y -122.2915,Z 152,A -111.1651,B 20.2003,C -0.5569,E1 20.1545,E2 199.1226} C_DIS
LIN {X -45.6304,Y -121.1739,Z 152,A -112.6454,B 20.2003,C -0.5571,E1 20.1506,E2 200.6061} C_DIS
LIN {X -52.8281,Y -118.2132,Z 152,A -116.0834,B 20.2002,C -0.5609,E1 20.1418,E2 204.043} C_DIS
LIN {X -57.5869,Y -115.97,Z 152,A -118.4418,B 20.2002,C -0.5625,E1 20.1358,E2 206.4045} C_DIS
LIN {X -61.5829,Y -113.9006,Z 152,A -120.5384,B 20.2002,C -0.5609,E1 20.1306,E2 208.5129} C_DIS
LIN {X -65.4992,Y -111.6939,Z 152,A -123.1534,B 20.2007,C -0.5396,E1 20.1241,E2 211.1998} C_DIS
LIN {X -70.1528,Y -108.832,Z 152,A -124.9312,B 20.2,C -0.5679,E1 20.1201,E2 212.9025} C_DIS
LIN {X -75.7682,Y -104.9996,Z 152,A -127.7436,B 20.1997,C -0.5803,E1 20.1137,E2 215.6907} C_DIS
LIN {X -78.1005,Y -103.2763,Z 152,A -129.2274,B 20.1998,C -0.5748,E1 20.1103,E2 217.1972} C_DIS
LIN {X -81.5704,Y -100.5588,Z 152,A -131.2249,B 20.1998,C -0.5766,E1 20.106,E2 219.1992} C_DIS
LIN {X -84.9426,Y -97.7266,Z 152,A -133.1781,B 20.1997,C -0.5801,E1 20.1018,E2 221.1517} C_DIS
LIN {X -88.9768,Y -94.0681,Z 152,A -135.9475,B 20.1999,C -0.5713,E1 20.0961,E2 223.961} C_DIS
LIN {X -91.8418,Y -91.2729,Z 152,A -137.1726,B 20.1992,C -0.5957,E1 20.0938,E2 225.1216} C_DIS
LIN {X -94.2389,Y -88.7958,Z 152,A -138.9367,B 20.1994,C -0.5899,E1 20.0903,E2 226.9123} C_DIS
LIN {X -96.9566,Y -85.8201,Z 152,A -140.6724,B 20.1992,C -0.5957,E1 20.0871,E2 228.641} C_DIS
LIN {X -99.834,Y -82.4552,Z 152,A -142.621,B 20.1991,C -0.6005,E1 20.0836,E2 230.5867} C_DIS
LIN {X -102.3314,Y -79.3344,Z 152,A -144.4246,B 20.1991,C -0.6034,E1 20.0805,E2 232.3928} C_DIS
LIN {X -104.9286,Y -75.8661,Z 152,A -146.3528,B 20.1989,C -0.6076,E1 20.0773,E2 234.3204} C_DIS
LIN {X -107.4457,Y -72.2581,Z 152,A -148.3719,B 20.1989,C -0.6098,E1 20.0741,E2 236.346} C_DIS
LIN {X -109.9808,Y -68.3367,Z 152,A -150.4165,B 20.1987,C -0.6159,E1 20.071,E2 238.386} C_DIS
LIN {X -112.1893,Y -64.6475,Z 152,A -152.7812,B 20.199,C -0.6037,E1 20.0676,E2 240.8018} C_DIS
LIN {X -114.3304,Y -60.7795,Z 152,A -154.125,B 20.1982,C -0.6317,E1 20.066,E2 242.0729} C_DIS
LIN {X -115.4951,Y -58.5328,Z 152,A -155.325,B 20.1982,C -0.6317,E1 20.0644,E2 243.2809} C_DIS
LIN {X -116.99,Y -55.4854,Z 152,A -156.8631,B 20.1981,C -0.6345,E1 20.0625,E2 244.8214} C_DIS
LIN {X -118.5031,Y -52.1793,Z 152,A -158.4368,B 20.1979,C -0.6403,E1 20.0607,E2 246.3891} C_DIS
LIN {X -119.6565,Y -49.4743,Z 152,A -159.7997,B 20.1979,C -0.6417,E1 20.0593,E2 247.7576} C_DIS
LIN {X -121.5363,Y -44.6627,Z 152,A -162.744,B 20.1984,C -0.624,E1 20.0563,E2 250.7745} C_DIS
LIN {X -123.1633,Y -39.9543,Z 152,A -164.1902,B 20.1974,C -0.6584,E1 20.0551,E2 252.1309} C_DIS
LIN {X -124.2519,Y -36.4237,Z 152,A -165.9755,B 20.1974,C -0.6577,E1 20.0536,E2 253.9313} C_DIS
LIN {X -125.2203,Y -32.9436,Z 152,A -167.5896,B 20.1973,C -0.6619,E1 20.0525,E2 255.5452} C_DIS
LIN {X -126.1251,Y -29.2899,Z 152,A -169.2897,B 20.1971,C -0.6656,E1 20.0514,E2 257.2469} C_DIS
LIN {X -126.8847,Y -25.7974,Z 152,A -170.819,B 20.1969,C -0.6724,E1 20.0505,E2 258.768} C_DIS
LIN {X -127.4609,Y -22.7811,Z 152,A -172.2786,B 20.1969,C -0.6728,E1 20.0497,E2 260.2372} C_DIS
LIN {X -128.1863,Y -18.263,Z 152,A -174.2366,B 20.1966,C -0.6815,E1 20.0489,E2 262.1846} C_DIS
LIN {X -128.923,Y -12.011,Z 152,A -176.8382,B 20.1961,C -0.6969,E1 20.0481,E2 264.7611} C_DIS
LIN {X -129.2419,Y -7.8636,Z 152,A -178.9396,B 20.1963,C -0.6931,E1 20.0477,E2 266.8897} C_DIS
LIN {X -129.4641,Y -2.0908,Z 152,A 178.5917,B 20.1959,C -0.7043,E1 20.0475,E2 269.3445} C_DIS
LIN {X -129.4787,Y 0.9048,Z 152,A 176.7589,B 20.1964,C -0.6899,E1 20.0475,E2 271.2333} C_DIS
LIN {X -129.3967,Y 4.6835,Z 152,A 175.5787,B 20.1956,C -0.7132,E1 20.0475,E2 272.3547} C_DIS
LIN {X -129.2248,Y 8.1414,Z 152,A 173.1562,B 20.1965,C -0.6856,E1 20.048,E2 274.8762} C_DIS
LIN {X -128.7456,Y 13.7785,Z 152,A 171.4136,B 20.1953,C -0.7211,E1 20.0485,E2 276.5284} C_DIS
LIN {X -128.3093,Y 17.3872,Z 152,A 169.7349,B 20.1953,C -0.7236,E1 20.0491,E2 278.2126} C_DIS
LIN {X -127.7154,Y 21.308,Z 152,A 168.0016,B 20.195,C -0.7299,E1 20.0498,E2 279.9407} C_DIS
LIN {X -126.9709,Y 25.3738,Z 152,A 166.1309,B 20.1949,C -0.734,E1 20.0508,E2 281.8132} C_DIS
LIN {X -126.1682,Y 29.1016,Z 152,A 164.4761,B 20.1946,C -0.7405,E1 20.0518,E2 283.4616} C_DIS
LIN {X -125.1574,Y 33.1797,Z 152,A 161.4415,B 20.1959,C -0.7036,E1 20.0541,E2 286.6262} C_DIS
LIN {X -123.0003,Y 40.452,Z 152,A 158.3943,B 20.1952,C -0.7249,E1 20.0567,E2 289.6333} C_DIS
LIN {X -121.0256,Y 46.0262,Z 152,A 156.4653,B 20.194,C -0.7578,E1 20.0585,E2 291.4804} C_DIS
LIN {X -119.1809,Y 50.6132,Z 152,A 154.4115,B 20.1936,C -0.7692,E1 20.0606,E2 293.5154} C_DIS
LIN {X -117.878,Y 53.5775,Z 152,A 152.7893,B 20.1937,C -0.7664,E1 20.0625,E2 295.1569} C_DIS
LIN {X -116.1488,Y 57.2242,Z 152,A 150.0064,B 20.1948,C -0.7353,E1 20.0661,E2 298.0494} C_DIS
LIN {X -112.6537,Y 63.8354,Z 152,A 148.0033,B 20.1928,C -0.7923,E1 20.0686,E2 299.8998} C_DIS
LIN {X -108.225,Y 71.0847,Z 152,A 143.9325,B 20.1928,C -0.7911,E1 20.0746,E2 304.0006} C_DIS
LIN {X -105.7001,Y 74.7877,Z 152,A 141.9383,B 20.1926,C -0.796,E1 20.0778,E2 305.993} C_DIS
LIN {X -103.0841,Y 78.3548,Z 152,A 139.9444,B 20.1925,C -0.7997,E1 20.0811,E2 307.9881} C_DIS
LIN {X -100.3812,Y 81.7882,Z 152,A 138.0514,B 20.1922,C -0.8062,E1 20.0844,E2 309.8735} C_DIS
LIN {X -97.7499,Y 84.9158,Z 152,A 136.168,B 20.1922,C -0.8079,E1 20.0878,E2 311.7628} C_DIS
LIN {X -94.673,Y 88.3329,Z 152,A 134.1417,B 20.192,C -0.8131,E1 20.0916,E2 313.7852} C_DIS
LIN {X -91.5883,Y 91.5281,Z 152,A 132.1754,B 20.1918,C -0.8177,E1 20.0955,E2 315.7488} C_DIS
LIN {X -88.5193,Y 94.4994,Z 152,A 130.2583,B 20.1917,C -0.821,E1 20.0994,E2 317.6663} C_DIS
LIN {X -85.3173,Y 97.3996,Z 152,A 128.3693,B 20.1915,C -0.8261,E1 20.1033,E2 319.55} C_DIS
LIN {X -82.1548,Y 100.0817,Z 152,A 126.4711,B 20.1915,C -0.8276,E1 20.1074,E2 321.453} C_DIS
LIN {X -78.5557,Y 102.9305,Z 152,A 124.4826,B 20.1912,C -0.8334,E1 20.1117,E2 323.4339} C_DIS
LIN {X -75.0204,Y 105.5355,Z 152,A 122.4758,B 20.1912,C -0.8348,E1 20.1163,E2 325.4455} C_DIS
LIN {X -71.9453,Y 107.6547,Z 152,A 120.3375,B 20.1917,C -0.8197,E1 20.1214,E2 327.6368} C_DIS
LIN {X -67.9594,Y 110.2147,Z 152,A 119.0543,B 20.1903,C -0.8541,E1 20.1242,E2 328.825} C_DIS
LIN {X -65.4988,Y 111.6941,Z 152,A 117.4754,B 20.1907,C -0.8446,E1 20.128,E2 330.4377} C_DIS
LIN {X -61.6212,Y 113.8798,Z 152,A 115.3931,B 20.1907,C -0.8436,E1 20.1332,E2 332.5305} C_DIS
LIN {X -57.899,Y 115.816,Z 152,A 113.648,B 20.1905,C -0.8507,E1 20.1375,E2 334.2608} C_DIS
LIN {X -54.5764,Y 117.4166,Z 152,A 111.3069,B 20.1915,C -0.8262,E1 20.1436,E2 336.6804} C_DIS
LIN {X -49.458,Y 119.6633,Z 152,A 110.1221,B 20.1893,C -0.8788,E1 20.1463,E2 337.7158} C_DIS
LIN {X -43.4886,Y 121.9596,Z 152,A 106.8105,B 20.19,C -0.8637,E1 20.155,E2 341.0802} C_DIS
LIN {X -40.738,Y 122.905,Z 152,A 105.4314,B 20.19,C -0.8616,E1 20.1587,E2 342.4687} C_DIS
LIN {X -36.6036,Y 124.1992,Z 152,A 103.5336,B 20.19,C -0.8644,E1 20.1637,E2 344.3625} C_DIS
LIN {X -33.0568,Y 125.1901,Z 152,A 101.9679,B 20.1898,C -0.8685,E1 20.1679,E2 345.9195} C_DIS
LIN {X -29.8873,Y 125.9849,Z 152,A 100.3276,B 20.19,C -0.8622,E1 20.1724,E2 347.5808} C_DIS
LIN {X -22.5328,Y 127.5053,Z 152,A 97.2277,B 20.1896,C -0.8734,E1 20.1809,E2 350.6526} C_DIS
LIN {X -19.8059,Y 127.957,Z 152,A 95.4239,B 20.1904,C -0.8515,E1 20.186,E2 352.5218} C_DIS
LIN {X -15.7154,Y 128.5238,Z 152,A 93.9324,B 20.1899,C -0.8656,E1 20.19,E2 353.9738} C_DIS
LIN {X -7.8392,Y 129.2434,Z 152,A 90.7221,B 20.1893,C -0.8785,E1 20.1989,E2 357.1487} C_DIS
LIN {X -5.0229,Y 129.3834,Z 152,A 88.6493,B 20.1907,C -0.8463,E1 20.2049,E2 359.3152} C_DIS
LIN {X 0.1234,Y 129.4823,Z 152,A 87.1429,B 20.1894,C -0.8771,E1 20.2089,E2 360.7325} C_DIS
LIN {X 6.7035,Y 129.3074,Z 152,A 84.0795,B 20.1896,C -0.8712,E1 20.2175,E2 363.812} C_DIS
LIN {X 13.4311,Y 128.783,Z 152,A 80.9709,B 20.1899,C -0.8659,E1 20.2262,E2 366.9336} C_DIS
LIN {X 18.5252,Y 128.1488,Z 152,A 78.8681,B 20.1896,C -0.8721,E1 20.2319,E2 369.0163} C_DIS
LIN {X 24.4483,Y 127.1516,Z 152,A 76.5556,B 20.1891,C -0.885,E1 20.2382,E2 371.2884} C_DIS
LIN {X 26.6253,Y 126.7156,Z 152,A 75.0657,B 20.1899,C -0.864,E1 20.2424,E2 372.8368} C_DIS
LIN {X 30.7049,Y 125.7878,Z 152,A 73.4372,B 20.1896,C -0.8719,E1 20.2468,E2 374.4393} C_DIS
LIN {X 33.9645,Y 124.9481,Z 152,A 71.8264,B 20.1899,C -0.866,E1 20.2512,E2 376.064} C_DIS
LIN {X 37.9177,Y 123.8041,Z 152,A 70.0988,B 20.1898,C -0.8685,E1 20.2557,E2 377.7807} C_DIS
LIN {X 41.0462,Y 122.8024,Z 152,A 68.6465,B 20.1898,C -0.8673,E1 20.2596,E2 379.2329} C_DIS
LIN {X 44.3424,Y 121.6518,Z 152,A 66.6825,B 20.1906,C -0.8488,E1 20.2649,E2 381.2452} C_DIS
LIN {X 47.8635,Y 120.31,Z 152,A 65.1869,B 20.1903,C -0.8541,E1 20.2687,E2 382.7213} C_DIS
LIN {X 52.9966,Y 118.1378,Z 152,A 62.9104,B 20.1901,C -0.8591,E1 20.2745,E2 384.9762} C_DIS
LIN {X 57.4764,Y 116.0245,Z 152,A 60.793,B 20.1901,C -0.8595,E1 20.2798,E2 387.0855} C_DIS
LIN {X 60.6506,Y 114.3981,Z 152,A 59.1663,B 20.1903,C -0.8554,E1 20.2839,E2 388.7183} C_DIS
LIN {X 66.1369,Y 111.3176,Z 152,A 56.2676,B 20.1906,C -0.8467,E1 20.2909,E2 391.6312} C_DIS
LIN {X 70.2874,Y 108.7447,Z 152,A 54.1344,B 20.1907,C -0.8445,E1 20.2959,E2 393.7621} C_DIS
LIN {X 73.0796,Y 106.8882,Z 152,A 52.792,B 20.1906,C -0.8479,E1 20.299,E2 395.0887} C_DIS
LIN {X 76.3187,Y 104.6006,Z 152,A 50.9469,B 20.1909,C -0.8412,E1 20.3032,E2 396.9452} C_DIS
LIN {X 79.7383,Y 102.0175,Z 152,A 49.0457,B 20.191,C -0.8375,E1 20.3074,E2 398.848} C_DIS
LIN {X 83.2752,Y 99.1509,Z 152,A 47.1049,B 20.191,C -0.8369,E1 20.3116,E2 400.7814} C_DIS
LIN {X 86.6289,Y 96.2352,Z 152,A 45.1111,B 20.1912,C -0.8318,E1 20.3158,E2 402.7796} C_DIS
LIN {X 90.8567,Y 92.2539,Z 152,A 42.6645,B 20.1912,C -0.8318,E1 20.3207,E2 405.2137} C_DIS
LIN {X 93.4848,Y 89.5896,Z 152,A 40.9269,B 20.1915,C -0.8247,E1 20.3241,E2 406.9621} C_DIS
LIN {X 96.2777,Y 86.5814,Z 152,A 39.0862,B 20.1917,C -0.8197,E1 20.3276,E2 408.8071} C_DIS
LIN {X 99.2548,Y 83.1514,Z 152,A 37.1245,B 20.1918,C -0.8171,E1 20.3311,E2 410.7648} C_DIS
LIN {X 102.2571,Y 79.4302,Z 152,A 35.2342,B 20.1916,C -0.8217,E1 20.3344,E2 412.6307} C_DIS
LIN {X 104.1481,Y 76.9347,Z 152,A 33.5934,B 20.1922,C -0.8074,E1 20.3372,E2 414.3027} C_DIS
LIN {X 108.087,Y 71.2939,Z 152,A 30.7054,B 20.1922,C -0.8065,E1 20.3417,E2 417.1753} C_DIS
LIN {X 109.986,Y 68.3284,Z 152,A 28.8021,B 20.1929,C -0.7877,E1 20.3446,E2 419.1205} C_DIS
LIN {X 111.7872,Y 65.3405,Z 152,A 27.5326,B 20.1926,C -0.7954,E1 20.3464,E2 420.3598} C_DIS
LIN {X 113.9006,Y 61.5829,Z 152,A 25.605,B 20.1929,C -0.7894,E1 20.349,E2 422.2918} C_DIS
LIN {X 115.7037,Y 58.1231,Z 152,A 23.4665,B 20.1937,C -0.767,E1 20.3517,E2 424.4802} C_DIS
LIN {X 117.588,Y 54.2056,Z 152,A 22.0654,B 20.1931,C -0.7841,E1 20.3533,E2 425.8226} C_DIS
LIN {X 119.415,Y 50.0526,Z 152,A 19.6646,B 20.1939,C -0.7615,E1 20.356,E2 428.2718} C_DIS
LIN {X 120.9191,Y 46.3052,Z 152,A 18.3919,B 20.1933,C -0.7785,E1 20.3572,E2 429.4867} C_DIS
LIN {X 122.3676,Y 42.3245,Z 152,A 16.4796,B 20.1935,C -0.7714,E1 20.359,E2 431.4058} C_DIS
LIN {X 123.4493,Y 39.059,Z 152,A 14.9781,B 20.1937,C -0.7678,E1 20.3603,E2 432.9067} C_DIS
LIN {X 124.5983,Y 35.2224,Z 152,A 13.1131,B 20.194,C -0.7585,E1 20.3618,E2 434.7851} C_DIS
LIN {X 125.6284,Y 31.3526,Z 152,A 11.3316,B 20.1942,C -0.7528,E1 20.363,E2 436.5701} C_DIS
LIN {X 126.5014,Y 27.6176,Z 152,A 9.1081,B 20.1952,C -0.7249,E1 20.3644,E2 438.8574} C_DIS
LIN {X 127.4723,Y 22.717,Z 152,A 7.6735,B 20.1942,C -0.7517,E1 20.3651,E2 440.2043} C_DIS
LIN {X 128.2265,Y 17.9816,Z 152,A 5.223,B 20.195,C -0.7309,E1 20.3661,E2 442.6966} C_DIS
LIN {X 129.1267,Y 9.5714,Z 152,A 1.8065,B 20.1949,C -0.7334,E1 20.3671,E2 446.0802} C_DIS
LIN {X 129.4564,Y 2.5504,Z 152,A -1.1599,B 20.195,C -0.7299,E1 20.3674,E2 449.0344} C_DIS
LIN {X 129.4399,Y -3.2741,Z 152,A -3.6877,B 20.1952,C -0.7239,E1 20.3674,E2 451.5604} C_DIS
LIN {X 129.3287,Y -6.2794,Z 152,A -5.2752,B 20.1957,C -0.7084,E1 20.3672,E2 453.1804} C_DIS
LIN {X 128.9193,Y -12.0502,Z 152,A -8.3499,B 20.1967,C -0.678,E1 20.3665,E2 456.3195} C_DIS
LIN {X 128.3956,Y -16.7288,Z 152,A -9.6834,B 20.1959,C -0.7041,E1 20.3661,E2 457.568} C_DIS
LIN {X 127.1705,Y -24.3497,Z 152,A -13.2086,B 20.1964,C -0.6885,E1 20.3644,E2 461.1119} C_DIS
LIN {X 126.4404,Y -27.9,Z 152,A -14.9025,B 20.1967,C -0.6796,E1 20.3634,E2 462.819} C_DIS
LIN {X 125.5018,Y -31.8516,Z 152,A -16.5973,B 20.1967,C -0.6785,E1 20.3623,E2 464.5045} C_DIS
LIN {X 124.6193,Y -35.1473,Z 152,A -18.0376,B 20.1967,C -0.6769,E1 20.3612,E2 465.939} C_DIS
LIN {X 123.7391,Y -38.1302,Z 152,A -19.4671,B 20.197,C -0.6703,E1 20.3601,E2 467.3771} C_DIS
LIN {X 122.4525,Y -42.0796,Z 152,A -21.3691,B 20.1973,C -0.6619,E1 20.3584,E2 469.2897} C_DIS
LIN {X 120.9755,Y -46.1599,Z 152,A -23.1541,B 20.1973,C -0.6619,E1 20.3567,E2 471.0618} C_DIS
LIN {X 119.1944,Y -50.5805,Z 152,A -25.232,B 20.1974,C -0.657,E1 20.3545,E2 473.1394} C_DIS
LIN {X 118.1464,Y -52.9774,Z 152,A -26.4135,B 20.1975,C -0.6526,E1 20.3531,E2 474.3255} C_DIS
LIN {X 116.758,Y -55.971,Z 152,A -28.7301,B 20.1988,C -0.6113,E1 20.3502,E2 476.7452} C_DIS
LIN {X 113.9572,Y -61.4775,Z 152,A -30.4644,B 20.1977,C -0.6466,E1 20.3481,E2 478.3664} C_DIS
LIN {X 112.2696,Y -64.5088,Z 152,A -32.215,B 20.1981,C -0.6329,E1 20.3456,E2 480.1449} C_DIS
LIN {X 110.0351,Y -68.2494,Z 152,A -34.1104,B 20.1983,C -0.6289,E1 20.3429,E2 482.0395} C_DIS
LIN {X 107.8872,Y -71.5972,Z 152,A -35.8256,B 20.1983,C -0.626,E1 20.3403,E2 483.7521} C_DIS
LIN {X 105.5457,Y -75.0061,Z 152,A -37.7126,B 20.1986,C -0.6187,E1 20.3373,E2 485.6487} C_DIS
LIN {X 102.7897,Y -78.7397,Z 152,A -39.6242,B 20.1986,C -0.6194,E1 20.3341,E2 487.5466} C_DIS
LIN {X 100.6306,Y -81.4814,Z 152,A -41.2698,B 20.1988,C -0.611,E1 20.3312,E2 489.2066} C_DIS
LIN {X 97.0713,Y -85.6903,Z 152,A -43.9318,B 20.1992,C -0.5953,E1 20.3263,E2 491.8985} C_DIS
LIN {X 94.7304,Y -88.2713,Z 152,A -45.0555,B 20.1988,C -0.6095,E1 20.3242,E2 492.975} C_DIS
LIN {X 92.2026,Y -90.9091,Z 152,A -46.7806,B 20.1991,C -0.601,E1 20.3208,E2 494.7154} C_DIS
LIN {X 88.27,Y -94.7316,Z 152,A -49.3518,B 20.1994,C -0.5892,E1 20.3156,E2 497.3071} C_DIS
LIN {X 85.5718,Y -97.1761,Z 152,A -50.8224,B 20.1994,C -0.5916,E1 20.3126,E2 498.7633} C_DIS
LIN {X 82.3065,Y -99.9571,Z 152,A -52.6643,B 20.1994,C -0.5899,E1 20.3086,E2 500.6012} C_DIS
LIN {X 77.1197,Y -104.011,Z 152,A -55.3174,B 20.1993,C -0.5949,E1 20.3029,E2 503.2273} C_DIS
LIN {X 73.2071,Y -106.8007,Z 152,A -57.7206,B 20.1997,C -0.5789,E1 20.2973,E2 505.6661} C_DIS
LIN {X 69.4652,Y -109.2722,Z 152,A -59.725,B 20.1998,C -0.5743,E1 20.2926,E2 507.6755} C_DIS
LIN {X 65.7271,Y -111.5601,Z 152,A -61.6389,B 20.1998,C -0.572,E1 20.288,E2 509.5887} C_DIS
LIN {X 61.7185,Y -113.8271,Z 152,A -63.6875,B 20.2,C -0.5681,E1 20.283,E2 511.6409} C_DIS
LIN {X 54.9022,Y -117.2659,Z 152,A -66.8406,B 20.1999,C -0.5722,E1 20.2752,E2 514.7711} C_DIS
LIN {X 45.8957,Y -121.0745,Z 152,A -71.2004,B 20.2001,C -0.5648,E1 20.2639,E2 519.1394} C_DIS
LIN {X 42.6061,Y -122.27,Z 152,A -72.8243,B 20.2002,C -0.5598,E1 20.2596,E2 520.7738} C_DIS
LIN {X 39.0196,Y -123.4619,Z 152,A -74.5338,B 20.2003,C -0.5563,E1 20.255,E2 522.4893} C_DIS
LIN {X 34.3299,Y -124.8479,Z 152,A -76.4701,B 20.2001,C -0.5635,E1 20.2499,E2 524.4006} C_DIS
LIN {X 31.4461,Y -125.6047,Z 152,A -78.0513,B 20.2004,C -0.5513,E1 20.2455,E2 526.014} C_DIS
LIN {X 24.6451,Y -127.114,Z 152,A -80.9421,B 20.2004,C -0.5566,E1 20.2377,E2 528.8846} C_DIS
LIN {X 20.5642,Y -127.8377,Z 152,A -83.0846,B 20.2007,C -0.5426,E1 20.2317,E2 531.0649} C_DIS
LIN {X 15.1845,Y -128.5874,Z 152,A -85.7612,B 20.201,C -0.53,E1 20.2242,E2 533.7751} C_DIS
LIN {X 10.8636,Y -129.0243,Z 152,A -87.4718,B 20.2008,C -0.5377,E1 20.2195,E2 535.4622} C_DIS
LIN {X 7.5227,Y -129.2629,Z 152,A -88.7588,B 20.2006,C -0.5451,E1 20.216,E2 536.7272} C_DIS
LIN {X 3.5748,Y -129.4316,Z 152,A -90.3945,B 20.2005,C -0.5492,E1 20.2114,E2 538.3506} C_DIS
LIN {X 0.921,Y -129.4737,Z 152,A -91.3607,B 20.2003,C -0.5575,E1 20.2088,E2 539.2926} C_DIS
Enddeposition()
LIN {X 0.921,Y -129.4737,Z 152,A -91.3607,B 20.2003,C -0.5575,E1 20.2088,E2 539.2926} C_DIS
Startdeposition()
$VEL.CP = VEL_PRINT
LIN {X 1.7436,Y -128.5279,Z 152,A -90.0677,B 18.8303,C -0.411,E1 18.8385,E2 538.3063} C_DIS
LIN {X 4.9858,Y -128.4423,Z 152,A -88.6564,B 18.8303,C -0.4101,E1 18.8424,E2 536.8982} C_DIS
LIN {X 7.7364,Y -128.3061,Z 152,A -86.2618,B 18.8293,C -0.4558,E1 18.8495,E2 534.3635} C_DIS
LIN {X 15.3255,Y -127.6221,Z 152,A -84.0125,B 18.8302,C -0.4129,E1 18.8553,E2 532.2494} C_DIS
LIN {X 18.9437,Y -127.1374,Z 152,A -81.9563,B 18.8298,C -0.4305,E1 18.8612,E2 530.1411} C_DIS
LIN {X 22.8086,Y -126.4991,Z 152,A -80.5483,B 18.8301,C -0.4186,E1 18.8649,E2 528.772} C_DIS
LIN {X 26.3516,Y -125.8103,Z 152,A -78.8729,B 18.8301,C -0.4225,E1 18.8695,E2 527.0876} C_DIS
LIN {X 30.9039,Y -124.7706,Z 152,A -76.8415,B 18.8301,C -0.4225,E1 18.875,E2 525.0605} C_DIS
LIN {X 35.3276,Y -123.5909,Z 152,A -74.7563,B 18.8299,C -0.4262,E1 18.8807,E2 522.9682} C_DIS
LIN {X 39.1735,Y -122.424,Z 152,A -73.1771,B 18.8301,C -0.4199,E1 18.8848,E2 521.4124} C_DIS
LIN {X 42.7941,Y -121.208,Z 152,A -71.427,B 18.83,C -0.4237,E1 18.8894,E2 519.6552} C_DIS
LIN {X 46.1636,Y -119.9637,Z 152,A -69.4974,B 18.8297,C -0.4388,E1 18.8946,E2 517.6849} C_DIS
LIN {X 49.504,Y -118.6235,Z 152,A -68.2151,B 18.8299,C -0.4282,E1 18.8978,E2 516.4392} C_DIS
LIN {X 53.3007,Y -116.9688,Z 152,A -66.3976,B 18.8299,C -0.4297,E1 18.9024,E2 514.6233} C_DIS
LIN {X 56.5846,Y -115.4142,Z 152,A -64.9028,B 18.8299,C -0.4272,E1 18.9062,E2 513.1416} C_DIS
LIN {X 62.0179,Y -112.59,Z 152,A -62.0107,B 18.8297,C -0.4381,E1 18.9133,E2 510.2272} C_DIS
LIN {X 66.0057,Y -110.2994,Z 152,A -59.9848,B 18.8297,C -0.4407,E1 18.9182,E2 508.2018} C_DIS
LIN {X 69.7446,Y -107.9742,Z 152,A -58.0083,B 18.8295,C -0.4448,E1 18.9229,E2 506.2213} C_DIS
LIN {X 73.5659,Y -105.4075,Z 152,A -56.0943,B 18.8295,C -0.4432,E1 18.9273,E2 504.3212} C_DIS
LIN {X 76.614,Y -103.2132,Z 152,A -54.5247,B 18.8295,C -0.4423,E1 18.9308,E2 502.7619} C_DIS
LIN {X 79.7961,Y -100.7737,Z 152,A -52.5144,B 18.8293,C -0.4549,E1 18.9353,E2 500.7228} C_DIS
LIN {X 83.1969,Y -97.9843,Z 152,A -50.5901,B 18.8293,C -0.4576,E1 18.9394,E2 498.8002} C_DIS
LIN {X 86.6577,Y -94.9381,Z 152,A -48.567,B 18.8292,C -0.4609,E1 18.9436,E2 496.7782} C_DIS
LIN {X 89.6824,Y -92.0861,Z 152,A -46.7789,B 18.8292,C -0.4625,E1 18.9472,E2 494.9953} C_DIS
LIN {X 92.5593,Y -89.1937,Z 152,A -44.991,B 18.829,C -0.4655,E1 18.9507,E2 493.2085} C_DIS
LIN {X 95.267,Y -86.2952,Z 152,A -43.1019,B 18.8288,C -0.4747,E1 18.9543,E2 491.3025} C_DIS
LIN {X 98.2133,Y -82.9274,Z 152,A -41.1328,B 18.8288,C -0.4786,E1 18.9579,E2 489.3336} C_DIS
LIN {X 100.8903,Y -79.6486,Z 152,A -39.2733,B 18.8286,C -0.4823,E1 18.9611,E2 487.4747} C_DIS
LIN {X 103.0935,Y -76.7749,Z 152,A -37.6991,B 18.8286,C -0.4848,E1 18.9638,E2 485.9029} C_DIS
LIN {X 105.5631,Y -73.3423,Z 152,A -35.8222,B 18.8285,C -0.4895,E1 18.9668,E2 484.0242} C_DIS
LIN {X 107.7121,Y -70.1484,Z 152,A -34.2615,B 18.8285,C -0.4877,E1 18.9692,E2 482.4794} C_DIS
LIN {X 109.7565,Y -66.9051,Z 152,A -32.396,B 18.8282,C -0.4988,E1 18.9719,E2 480.5927} C_DIS
LIN {X 111.9351,Y -63.1922,Z 152,A -30.5811,B 18.8282,C -0.4999,E1 18.9745,E2 478.7873} C_DIS
LIN {X 113.2442,Y -60.8145,Z 152,A -29.0941,B 18.8278,C -0.5147,E1 18.9765,E2 477.2655} C_DIS
LIN {X 115.6581,Y -56.0885,Z 152,A -26.9417,B 18.8278,C -0.5127,E1 18.9791,E2 475.1349} C_DIS
LIN {X 117.2679,Y -52.6349,Z 152,A -25.4348,B 18.8279,C -0.5098,E1 18.9808,E2 473.6481} C_DIS
LIN {X 118.5854,Y -49.5951,Z 152,A -23.8436,B 18.8277,C -0.5188,E1 18.9826,E2 472.0411} C_DIS
LIN {X 120.0149,Y -46.0318,Z 152,A -21.656,B 18.827,C -0.5435,E1 18.9849,E2 469.7942} C_DIS
LIN {X 121.5484,Y -41.8123,Z 152,A -20.1405,B 18.8274,C -0.5294,E1 18.9862,E2 468.3335} C_DIS
LIN {X 122.8046,Y -37.9652,Z 152,A -18.3913,B 18.8274,C -0.5326,E1 18.9877,E2 466.588} C_DIS
LIN {X 123.8829,Y -34.2835,Z 152,A -16.6627,B 18.8272,C -0.5386,E1 18.989,E2 464.8546} C_DIS
LIN {X 124.7663,Y -30.9209,Z 152,A -15.1717,B 18.8272,C -0.5409,E1 18.99,E2 463.3683} C_DIS
LIN {X 125.6543,Y -27.0782,Z 152,A -13.5274,B 18.8271,C -0.5416,E1 18.991,E2 461.7347} C_DIS
LIN {X 126.159,Y -24.6248,Z 152,A -12.3024,B 18.8269,C -0.5495,E1 18.9917,E2 460.4952} C_DIS
LIN {X 127.1223,Y -19.0414,Z 152,A -9.8652,B 18.8267,C -0.5537,E1 18.9928,E2 458.0647} C_DIS
LIN {X 127.5656,Y -15.7988,Z 152,A -8.3957,B 18.8267,C -0.5587,E1 18.9933,E2 456.5917} C_DIS
LIN {X 127.961,Y -12.1762,Z 152,A -6.7756,B 18.8265,C -0.5636,E1 18.9938,E2 454.9697} C_DIS
LIN {X 128.4085,Y -5.8259,Z 152,A -4.037,B 18.8263,C -0.5683,E1 18.9943,E2 452.2387} C_DIS
LIN {X 128.5238,Y 1.9914,Z 152,A -0.0839,B 18.8254,C -0.5984,E1 18.9943,E2 448.2251} C_DIS
LIN {X 128.4015,Y 5.9476,Z 152,A 1.3858,B 18.8256,C -0.5917,E1 18.9941,E2 446.788} C_DIS
LIN {X 128.1031,Y 10.5799,Z 152,A 4.1637,B 18.8245,C -0.6274,E1 18.9935,E2 443.9228} C_DIS
LIN {X 127.4426,Y 16.752,Z 152,A 6.3171,B 18.8251,C -0.6105,E1 18.9928,E2 441.8388} C_DIS
LIN {X 126.9777,Y 19.9751,Z 152,A 7.4494,B 18.8253,C -0.6018,E1 18.9923,E2 440.7422} C_DIS
LIN {X 126.3486,Y 23.6332,Z 152,A 8.9612,B 18.8253,C -0.601,E1 18.9916,E2 439.2451} C_DIS
LIN {X 125.6471,Y 27.1114,Z 152,A 10.5407,B 18.8253,C -0.6057,E1 18.9907,E2 437.6637} C_DIS
LIN {X 124.9691,Y 30.0823,Z 152,A 12.0733,B 18.8249,C -0.6169,E1 18.9897,E2 436.1089} C_DIS
LIN {X 123.8374,Y 34.4461,Z 152,A 13.8394,B 18.8249,C -0.6129,E1 18.9884,E2 434.3688} C_DIS
LIN {X 123.1589,Y 36.8048,Z 152,A 15.2091,B 18.8245,C -0.6273,E1 18.9873,E2 432.9655} C_DIS
LIN {X 122.0222,Y 40.408,Z 152,A 16.7711,B 18.8245,C -0.6273,E1 18.986,E2 431.4156} C_DIS
LIN {X 120.8042,Y 43.9163,Z 152,A 18.5183,B 18.8242,C -0.6358,E1 18.9843,E2 429.6556} C_DIS
LIN {X 118.591,Y 49.5816,Z 152,A 21.116,B 18.8242,C -0.6388,E1 18.9816,E2 427.0682} C_DIS
LIN {X 117.0325,Y 53.1611,Z 152,A 22.7945,B 18.8241,C -0.6411,E1 18.9797,E2 425.395} C_DIS
LIN {X 114.8639,Y 57.6968,Z 152,A 25.1378,B 18.8237,C -0.6514,E1 18.9769,E2 423.0373} C_DIS
LIN {X 113.0834,Y 61.1139,Z 152,A 26.8594,B 18.8236,C -0.6561,E1 18.9746,E2 421.3135} C_DIS
LIN {X 111.1128,Y 64.6271,Z 152,A 28.4221,B 18.8237,C -0.6515,E1 18.9725,E2 419.7763} C_DIS
LIN {X 109.0749,Y 68.0098,Z 152,A 30.3082,B 18.8234,C -0.6611,E1 18.9697,E2 417.8738} C_DIS
LIN {X 106.6462,Y 71.7591,Z 152,A 32.7369,B 18.8226,C -0.6837,E1 18.9659,E2 415.3918} C_DIS
LIN {X 104.2881,Y 75.145,Z 152,A 34.2109,B 18.823,C -0.6735,E1 18.9635,E2 413.9592} C_DIS
LIN {X 101.7632,Y 78.5301,Z 152,A 36.0599,B 18.8229,C -0.6766,E1 18.9604,E2 412.1124} C_DIS
LIN {X 99.2041,Y 81.7392,Z 152,A 37.8973,B 18.8227,C -0.6812,E1 18.9572,E2 410.2726} C_DIS
LIN {X 96.3576,Y 85.0757,Z 152,A 39.8058,B 18.8227,C -0.6837,E1 18.9537,E2 408.368} C_DIS
LIN {X 93.4629,Y 88.2459,Z 152,A 41.6974,B 18.8225,C -0.687,E1 18.9501,E2 406.4776} C_DIS
LIN {X 90.3225,Y 91.4584,Z 152,A 43.6776,B 18.8224,C -0.6903,E1 18.9462,E2 404.4987} C_DIS
LIN {X 87.3302,Y 94.3198,Z 152,A 45.5284,B 18.8223,C -0.6943,E1 18.9424,E2 402.6461} C_DIS
LIN {X 84.3935,Y 96.9557,Z 152,A 47.215,B 18.8223,C -0.6949,E1 18.9389,E2 400.9669} C_DIS
LIN {X 81.4715,Y 99.4237,Z 152,A 48.988,B 18.822,C -0.7008,E1 18.9351,E2 399.185} C_DIS
LIN {X 77.8831,Y 102.2592,Z 152,A 51.0086,B 18.822,C -0.7037,E1 18.9306,E2 397.1655} C_DIS
LIN {X 74.3791,Y 104.8357,Z 152,A 52.916,B 18.8218,C -0.7058,E1 18.9263,E2 395.2609} C_DIS
LIN {X 71.6173,Y 106.7413,Z 152,A 54.6183,B 18.8215,C -0.7163,E1 18.9223,E2 393.5339} C_DIS
LIN {X 67.2045,Y 109.5728,Z 152,A 56.702,B 18.8217,C -0.71,E1 18.9175,E2 391.4788} C_DIS
LIN {X 61.2669,Y 113.0005,Z 152,A 59.8387,B 18.8214,C -0.7174,E1 18.9098,E2 388.3321} C_DIS
LIN {X 57.3415,Y 115.0408,Z 152,A 61.5443,B 18.8217,C -0.7096,E1 18.9056,E2 386.6568} C_DIS
LIN {X 54.0848,Y 116.6062,Z 152,A 63.4275,B 18.8212,C -0.7221,E1 18.9008,E2 384.7417} C_DIS
LIN {X 50.0636,Y 118.3897,Z 152,A 65.3425,B 18.8212,C -0.7225,E1 18.8959,E2 382.8319} C_DIS
LIN {X 42.8572,Y 121.1861,Z 152,A 68.8043,B 18.8211,C -0.7264,E1 18.8869,E2 379.3681} C_DIS
LIN {X 39.3049,Y 122.382,Z 152,A 70.3333,B 18.8212,C -0.7224,E1 18.8828,E2 377.8554} C_DIS
LIN {X 35.294,Y 123.6003,Z 152,A 72.1963,B 18.8212,C -0.7236,E1 18.8779,E2 375.9933} C_DIS
LIN {X 31.5181,Y 124.6147,Z 152,A 73.9828,B 18.8211,C -0.7264,E1 18.873,E2 374.2019} C_DIS
LIN {X 27.4928,Y 125.5648,Z 152,A 75.5908,B 18.8214,C -0.7185,E1 18.8687,E2 372.6213} C_DIS
LIN {X 24.1551,Y 126.2488,Z 152,A 77.1126,B 18.8214,C -0.7194,E1 18.8646,E2 371.0995} C_DIS
LIN {X 20.9547,Y 126.8195,Z 152,A 78.7819,B 18.821,C -0.7282,E1 18.8599,E2 369.4052} C_DIS
LIN {X 17.4782,Y 127.3468,Z 152,A 80.3321,B 18.821,C -0.7281,E1 18.8556,E2 367.8574} C_DIS
LIN {X 13.5688,Y 127.8209,Z 152,A 82.2034,B 18.8208,C -0.7328,E1 18.8504,E2 365.9733} C_DIS
LIN {X 7.1882,Y 128.3399,Z 152,A 85.0472,B 18.8208,C -0.7327,E1 18.8425,E2 363.1318} C_DIS
LIN {X 1.1594,Y 128.5347,Z 152,A 87.4508,B 18.8213,C -0.7219,E1 18.8359,E2 360.7623} C_DIS
LIN {X -6.9623,Y 128.3514,Z 152,A 91.1967,B 18.8211,C -0.7256,E1 18.8254,E2 357.0042} C_DIS
LIN {X -13.243,Y 127.856,Z 152,A 94.1756,B 18.8209,C -0.7308,E1 18.817,E2 354.0074} C_DIS
LIN {X -19.4884,Y 127.0531,Z 152,A 96.8625,B 18.8211,C -0.7248,E1 18.8096,E2 351.3362} C_DIS
LIN {X -23.1167,Y 126.444,Z 152,A 98.5327,B 18.8211,C -0.7248,E1 18.805,E2 349.6638} C_DIS
LIN {X -25.8678,Y 125.9093,Z 152,A 100.2068,B 18.8206,C -0.7394,E1 18.8003,E2 347.9417} C_DIS
LIN {X -29.7721,Y 125.0439,Z 152,A 101.5598,B 18.8212,C -0.7222,E1 18.7968,E2 346.6397} C_DIS
LIN {X -32.7429,Y 124.2991,Z 152,A 102.8917,B 18.8213,C -0.7198,E1 18.7932,E2 345.3127} C_DIS
LIN {X -36.3654,Y 123.2876,Z 152,A 104.661,B 18.8213,C -0.7215,E1 18.7884,E2 343.5342} C_DIS
LIN {X -40.3648,Y 122.0366,Z 152,A 106.4746,B 18.8214,C -0.7175,E1 18.7836,E2 341.7285} C_DIS
LIN {X -42.9523,Y 121.1518,Z 152,A 108.0236,B 18.821,C -0.728,E1 18.7795,E2 340.1428} C_DIS
LIN {X -46.0853,Y 119.9941,Z 152,A 109.1706,B 18.8215,C -0.7138,E1 18.7766,E2 339.0365} C_DIS
LIN {X -49.5251,Y 118.6146,Z 152,A 110.8622,B 18.8215,C -0.7131,E1 18.7722,E2 337.3419} C_DIS
LIN {X -53.8569,Y 116.7116,Z 152,A 112.8223,B 18.8219,C -0.7049,E1 18.7672,E2 335.4011} C_DIS
LIN {X -56.0862,Y 115.6592,Z 152,A 114.0387,B 18.8218,C -0.7074,E1 18.7641,E2 334.1725} C_DIS
LIN {X -59.359,Y 114.0125,Z 152,A 115.5351,B 18.822,C -0.7001,E1 18.7605,E2 332.6935} C_DIS
LIN {X -62.3254,Y 112.4198,Z 152,A 117.6042,B 18.8214,C -0.7179,E1 18.7552,E2 330.5609} C_DIS
LIN {X -65.554,Y 110.5686,Z 152,A 118.914,B 18.822,C -0.7026,E1 18.7522,E2 329.2931} C_DIS
LIN {X -71.5814,Y 106.7652,Z 152,A 122.4914,B 18.8217,C -0.7111,E1 18.7437,E2 325.6736} C_DIS
LIN {X -74.7199,Y 104.5925,Z 152,A 123.8414,B 18.8222,C -0.6954,E1 18.7407,E2 324.3661} C_DIS
LIN {X -78.2922,Y 101.9463,Z 152,A 125.8312,B 18.8223,C -0.6918,E1 18.7363,E2 322.3779} C_DIS
LIN {X -81.4303,Y 99.4574,Z 152,A 127.5743,B 18.8225,C -0.6866,E1 18.7325,E2 320.6419} C_DIS
LIN {X -84.4565,Y 96.9008,Z 152,A 129.3827,B 18.8226,C -0.6844,E1 18.7287,E2 318.8309} C_DIS
LIN {X -87.4459,Y 94.212,Z 152,A 131.2429,B 18.8226,C -0.6828,E1 18.7248,E2 316.9653} C_DIS
LIN {X -90.5823,Y 91.2003,Z 152,A 133.1571,B 18.8228,C -0.6776,E1 18.721,E2 315.0565} C_DIS
LIN {X -93.4848,Y 88.2226,Z 152,A 134.9868,B 18.823,C -0.6724,E1 18.7175,E2 313.2321} C_DIS
LIN {X -96.1504,Y 85.3101,Z 152,A 136.8375,B 18.823,C -0.6713,E1 18.714,E2 311.3734} C_DIS
LIN {X -99.1011,Y 81.8636,Z 152,A 138.7943,B 18.8233,C -0.6641,E1 18.7105,E2 309.427} C_DIS
LIN {X -101.56,Y 78.7922,Z 152,A 140.6475,B 18.8233,C -0.6631,E1 18.7073,E2 307.565} C_DIS
LIN {X -104.3075,Y 75.1182,Z 152,A 142.6756,B 18.8235,C -0.6572,E1 18.704,E2 305.5418} C_DIS
LIN {X -106.7563,Y 71.5947,Z 152,A 144.4578,B 18.8239,C -0.6476,E1 18.7012,E2 303.7773} C_DIS
LIN {X -109.8779,Y 66.705,Z 152,A 147.2329,B 18.8239,C -0.6471,E1 18.6971,E2 300.9843} C_DIS
LIN {X -112.2324,Y 62.6632,Z 152,A 149.3477,B 18.824,C -0.6424,E1 18.6941,E2 298.8693} C_DIS
LIN {X -115.2,Y 57.0188,Z 152,A 152.0658,B 18.8244,C -0.6301,E1 18.6907,E2 296.1697} C_DIS
LIN {X -116.4361,Y 54.4527,Z 152,A 153.307,B 18.8246,C -0.6255,E1 18.6892,E2 294.9337} C_DIS
LIN {X -117.8915,Y 51.2231,Z 152,A 154.9497,B 18.8246,C -0.6231,E1 18.6873,E2 293.286} C_DIS
LIN {X -119.4662,Y 47.4388,Z 152,A 156.9713,B 18.8246,C -0.6244,E1 18.6852,E2 291.245} C_DIS
LIN {X -121.3444,Y 42.4008,Z 152,A 159.2006,B 18.825,C -0.6116,E1 18.6831,E2 289.0385} C_DIS
LIN {X -122.3472,Y 39.4138,Z 152,A 160.7286,B 18.825,C -0.6116,E1 18.6817,E2 287.4985} C_DIS
LIN {X -123.4996,Y 35.6411,Z 152,A 162.3002,B 18.8254,C -0.5999,E1 18.6805,E2 285.951} C_DIS
LIN {X -124.85,Y 30.5762,Z 152,A 164.7815,B 18.8254,C -0.5977,E1 18.6788,E2 283.4567} C_DIS
LIN {X -125.727,Y 26.7411,Z 152,A 166.5524,B 18.8256,C -0.5929,E1 18.6777,E2 281.6864} C_DIS
LIN {X -126.5527,Y 22.5093,Z 152,A 168.5057,B 18.8257,C -0.5881,E1 18.6767,E2 279.7325} C_DIS
LIN {X -127.1878,Y 18.5926,Z 152,A 170.1378,B 18.826,C -0.5779,E1 18.676,E2 278.1187} C_DIS
LIN {X -127.5509,Y 15.9223,Z 152,A 171.6258,B 18.8259,C -0.584,E1 18.6754,E2 276.5996} C_DIS
LIN {X -127.9534,Y 12.2557,Z 152,A 173.355,B 18.8259,C -0.5818,E1 18.675,E2 274.863} C_DIS
LIN {X -128.2701,Y 8.3211,Z 152,A 174.9814,B 18.8262,C -0.5718,E1 18.6746,E2 273.2546} C_DIS
LIN {X -128.4764,Y 4.0426,Z 152,A 176.9315,B 18.8264,C -0.5672,E1 18.6744,E2 271.3026} C_DIS
LIN {X -128.5406,Y -0.312,Z 152,A 178.665,B 18.8267,C -0.5541,E1 18.6744,E2 269.5958} C_DIS
LIN {X -128.512,Y -2.6971,Z 152,A 179.985,B 18.8266,C -0.5596,E1 18.6744,E2 268.2478} C_DIS
LIN {X -128.3608,Y -6.7752,Z 152,A -178.1712,B 18.8267,C -0.5548,E1 18.6747,E2 266.4037} C_DIS
LIN {X -128.1192,Y -10.3886,Z 152,A -176.8307,B 18.8271,C -0.5404,E1 18.675,E2 265.097} C_DIS
LIN {X -127.7979,Y -13.7828,Z 152,A -175.0163,B 18.827,C -0.5459,E1 18.6755,E2 263.2507} C_DIS
LIN {X -127.2947,Y -17.8444,Z 152,A -173.276,B 18.8272,C -0.5374,E1 18.6761,E2 261.5226} C_DIS
LIN {X -126.757,Y -21.3295,Z 152,A -171.6937,B 18.8273,C -0.533,E1 18.6768,E2 259.9412} C_DIS
LIN {X -126.0154,Y -25.3462,Z 152,A -169.8673,B 18.8275,C -0.5277,E1 18.6778,E2 258.1165} C_DIS
LIN {X -125.2845,Y -28.7409,Z 152,A -168.3603,B 18.8276,C -0.5216,E1 18.6787,E2 256.6163} C_DIS
LIN {X -124.6186,Y -31.5028,Z 152,A -167.0543,B 18.8276,C -0.5192,E1 18.6796,E2 255.3074} C_DIS
LIN {X -123.849,Y -34.4045,Z 152,A -165.6904,B 18.8278,C -0.5162,E1 18.6806,E2 253.9422} C_DIS
LIN {X -122.6777,Y -38.3794,Z 152,A -163.5231,B 18.8276,C -0.5218,E1 18.6824,E2 251.7402} C_DIS
LIN {X -120.8368,Y -43.826,Z 152,A -161.1343,B 18.828,C -0.5084,E1 18.6846,E2 249.3746} C_DIS
LIN {X -119.5304,Y -47.2781,Z 152,A -159.611,B 18.8282,C -0.4995,E1 18.6861,E2 247.8674} C_DIS
LIN {X -118.2186,Y -50.4665,Z 152,A -158.1447,B 18.8284,C -0.4928,E1 18.6877,E2 246.411} C_DIS
LIN {X -116.7714,Y -53.7276,Z 152,A -156.6206,B 18.8285,C -0.4861,E1 18.6894,E2 244.8963} C_DIS
LIN {X -115.3792,Y -56.6555,Z 152,A -155.0124,B 18.8285,C -0.4878,E1 18.6914,E2 243.2707} C_DIS
LIN {X -113.9944,Y -59.3936,Z 152,A -153.7811,B 18.8287,C -0.4794,E1 18.6929,E2 242.0567} C_DIS
LIN {X -112.2904,Y -62.5591,Z 152,A -151.8804,B 18.8286,C -0.4855,E1 18.6955,E2 240.1232} C_DIS
LIN {X -110.0922,Y -66.3506,Z 152,A -149.9313,B 18.8286,C -0.4803,E1 18.6983,E2 238.1766} C_DIS
LIN {X -108.1783,Y -69.4272,Z 152,A -148.3065,B 18.8288,C -0.4766,E1 18.7007,E2 236.5521} C_DIS
LIN {X -105.7291,Y -73.1036,Z 152,A -146.3119,B 18.8288,C -0.4726,E1 18.7038,E2 234.5564} C_DIS
LIN {X -103.2352,Y -76.5845,Z 152,A -144.4026,B 18.829,C -0.468,E1 18.707,E2 232.6488} C_DIS
LIN {X -100.6055,Y -80.0074,Z 152,A -142.4702,B 18.829,C -0.4638,E1 18.7103,E2 230.7169} C_DIS
LIN {X -97.9522,Y -83.2347,Z 152,A -140.6151,B 18.8292,C -0.4593,E1 18.7136,E2 228.8642} C_DIS
LIN {X -95.0492,Y -86.5352,Z 152,A -138.8711,B 18.8295,C -0.4474,E1 18.7168,E2 227.1467} C_DIS
LIN {X -92.3113,Y -89.4498,Z 152,A -136.3737,B 18.829,C -0.4691,E1 18.7218,E2 224.567} C_DIS
LIN {X -89.1774,Y -92.575,Z 152,A -134.3684,B 18.829,C -0.4662,E1 18.7258,E2 222.5592} C_DIS
LIN {X -85.8879,Y -95.6344,Z 152,A -132.8233,B 18.8295,C -0.4459,E1 18.7289,E2 221.0689} C_DIS
LIN {X -82.7274,Y -98.3811,Z 152,A -130.941,B 18.8295,C -0.4429,E1 18.7329,E2 219.1858} C_DIS
LIN {X -79.1682,Y -101.2676,Z 152,A -128.8884,B 18.8296,C -0.4396,E1 18.7374,E2 217.1332} C_DIS
LIN {X -76.091,Y -103.5993,Z 152,A -127.4031,B 18.8299,C -0.4282,E1 18.7406,E2 215.6762} C_DIS
LIN {X -73.1517,Y -105.6957,Z 152,A -125.5105,B 18.8297,C -0.4357,E1 18.745,E2 213.7512} C_DIS
LIN {X -69.4825,Y -108.1429,Z 152,A -123.643,B 18.8299,C -0.4291,E1 18.7494,E2 211.8959} C_DIS
LIN {X -66.5387,Y -109.9784,Z 152,A -121.8266,B 18.8297,C -0.4367,E1 18.7538,E2 210.0483} C_DIS
LIN {X -61.8961,Y -112.6574,Z 152,A -119.6151,B 18.8299,C -0.4269,E1 18.7591,E2 207.8584} C_DIS
LIN {X -59.0177,Y -114.1914,Z 152,A -118.1269,B 18.8299,C -0.4263,E1 18.7628,E2 206.3666} C_DIS
LIN {X -54.5426,Y -116.3945,Z 152,A -115.9315,B 18.83,C -0.4227,E1 18.7683,E2 204.1748} C_DIS
LIN {X -50.8473,Y -118.054,Z 152,A -114.3191,B 18.8302,C -0.4136,E1 18.7724,E2 202.5853} C_DIS
LIN {X -45.8417,Y -120.0888,Z 152,A -111.6677,B 18.8301,C -0.4201,E1 18.7793,E2 199.9057} C_DIS
LIN {X -42.2062,Y -121.4118,Z 152,A -110.0393,B 18.8301,C -0.4151,E1 18.7836,E2 198.2885} C_DIS
LIN {X -38.3235,Y -122.695,Z 152,A -108.1975,B 18.8301,C -0.4144,E1 18.7885,E2 196.4445} C_DIS
LIN {X -34.5563,Y -123.8066,Z 152,A -106.5166,B 18.8303,C -0.4106,E1 18.793,E2 194.7717} C_DIS
LIN {X -31.2762,Y -124.6761,Z 152,A -104.9799,B 18.8303,C -0.4106,E1 18.7971,E2 193.232} C_DIS
LIN {X -27.2976,Y -125.6069,Z 152,A -103.3607,B 18.8305,C -0.4021,E1 18.8015,E2 191.6362} C_DIS
LIN {X -23.3086,Y -126.4097,Z 152,A -101.3167,B 18.8303,C -0.4099,E1 18.8072,E2 189.5649} C_DIS
LIN {X -19.6764,Y -127.024,Z 152,A -99.7071,B 18.8303,C -0.4082,E1 18.8116,E2 187.9586} C_DIS
LIN {X -16.0881,Y -127.5296,Z 152,A -98.2006,B 18.8304,C -0.4037,E1 18.8157,E2 186.4645} C_DIS
LIN {X -10.9369,Y -128.0729,Z 152,A -95.9058,B 18.8304,C -0.4029,E1 18.8221,E2 184.1706} C_DIS
LIN {X -3.887,Y -128.4807,Z 152,A -92.8312,B 18.8304,C -0.4001,E1 18.8307,E2 181.1034} C_DIS
LIN {X -0.5285,Y -128.5382,Z 152,A -91.018,B 18.8302,C -0.4123,E1 18.8358,E2 179.2522} C_DIS
LIN {X -0.5285,Y -128.5382,Z 152,A -91.018,B 18.8302,C -0.4123,E1 18.8358,E2 179.2522} C_DIS
Enddeposition()
LIN {X 0.9105,Y -127.5933,Z 152,A -90.4612,B 17.5246,C -0.2547,E1 17.528,E2 179.0895} C_DIS
Startdeposition()
$VEL.CP = VEL_PRINT
LIN {X -1.569,Y -127.5888,Z 152,A -91.8244,B 17.5247,C -0.2458,E1 17.5241,E2 180.4823} C_DIS
LIN {X -4.1048,Y -127.5324,Z 152,A -93.1241,B 17.5247,C -0.2401,E1 17.5204,E2 181.8009} C_DIS
LIN {X -7.8459,Y -127.3557,Z 152,A -94.6489,B 17.5247,C -0.2456,E1 17.5162,E2 183.3083} C_DIS
LIN {X -10.7592,Y -127.1427,Z 152,A -96.0324,B 17.5247,C -0.2432,E1 17.5124,E2 184.7006} C_DIS
LIN {X -14.0948,Y -126.817,Z 152,A -97.4939,B 17.5247,C -0.2449,E1 17.5083,E2 186.1577} C_DIS
LIN {X -17.0185,Y -126.4578,Z 152,A -98.819,B 17.5247,C -0.2451,E1 17.5046,E2 187.4834} C_DIS
LIN {X -20.1039,Y -126.0047,Z 152,A -100.2132,B 17.5247,C -0.2457,E1 17.5008,E2 188.8774} C_DIS
LIN {X -22.6364,Y -125.5732,Z 152,A -101.3952,B 17.5247,C -0.2452,E1 17.4975,E2 190.0629} C_DIS
LIN {X -26.2583,Y -124.8678,Z 152,A -103.1094,B 17.5247,C -0.2439,E1 17.4928,E2 191.7841} C_DIS
LIN {X -29.2469,Y -124.2017,Z 152,A -104.5053,B 17.5247,C -0.2439,E1 17.489,E2 193.1827} C_DIS
LIN {X -32.5219,Y -123.3833,Z 152,A -105.9428,B 17.5247,C -0.2475,E1 17.4852,E2 194.6113} C_DIS
LIN {X -35.5384,Y -122.5483,Z 152,A -107.291,B 17.5247,C -0.2504,E1 17.4815,E2 195.9531} C_DIS
LIN {X -38.3598,Y -121.6952,Z 152,A -108.5872,B 17.5247,C -0.2523,E1 17.4781,E2 197.2462} C_DIS
LIN {X -41.3408,Y -120.715,Z 152,A -110.0556,B 17.5247,C -0.2514,E1 17.4742,E2 198.7215} C_DIS
LIN {X -43.719,Y -119.8741,Z 152,A -111.3991,B 17.5247,C -0.2453,E1 17.4706,E2 200.0891} C_DIS
LIN {X -47.3982,Y -118.4671,Z 152,A -112.9817,B 17.5247,C -0.2533,E1 17.4665,E2 201.6503} C_DIS
LIN {X -50.1194,Y -117.3426,Z 152,A -114.3169,B 17.5246,C -0.2542,E1 17.4631,E2 202.987} C_DIS
LIN {X -52.425,Y -116.33,Z 152,A -115.5465,B 17.5246,C -0.2522,E1 17.4599,E2 204.2278} C_DIS
LIN {X -55.3386,Y -114.9726,Z 152,A -116.9692,B 17.5246,C -0.2545,E1 17.4564,E2 205.6478} C_DIS
LIN {X -58.6043,Y -113.345,Z 152,A -118.5601,B 17.5246,C -0.2581,E1 17.4524,E2 207.2332} C_DIS
LIN {X -61.2004,Y -111.964,Z 152,A -119.7834,B 17.5245,C -0.263,E1 17.4494,E2 208.445} C_DIS
LIN {X -64.2728,Y -110.2297,Z 152,A -121.4495,B 17.5245,C -0.2625,E1 17.4454,E2 210.1201} C_DIS
LIN {X -66.7697,Y -108.7347,Z 152,A -122.785,B 17.5245,C -0.2635,E1 17.4422,E2 211.4585} C_DIS
LIN {X -69.5847,Y -106.9551,Z 152,A -124.2815,B 17.5245,C -0.2657,E1 17.4386,E2 212.9546} C_DIS
LIN {X -72.1806,Y -105.2206,Z 152,A -125.6881,B 17.5245,C -0.2678,E1 17.4354,E2 214.3613} C_DIS
LIN {X -74.3031,Y -103.7327,Z 152,A -126.9651,B 17.5245,C -0.266,E1 17.4325,E2 215.6508} C_DIS
LIN {X -76.8508,Y -101.8595,Z 152,A -128.3698,B 17.5244,C -0.2689,E1 17.4293,E2 217.0531} C_DIS
LIN {X -80.2769,Y -99.182,Z 152,A -130.2539,B 17.5244,C -0.2746,E1 17.4252,E2 218.9285} C_DIS
LIN {X -82.7527,Y -97.1258,Z 152,A -131.8441,B 17.5244,C -0.2726,E1 17.4218,E2 220.5345} C_DIS
LIN {X -85.7532,Y -94.487,Z 152,A -133.6582,B 17.5243,C -0.2754,E1 17.418,E2 222.3499} C_DIS
LIN {X -89.1338,Y -91.3053,Z 152,A -135.7545,B 17.5243,C -0.2792,E1 17.4138,E2 224.4463} C_DIS
LIN {X -92.3469,Y -88.0539,Z 152,A -137.6909,B 17.5241,C -0.2872,E1 17.41,E2 226.3682} C_DIS
LIN {X -95.0117,Y -85.1715,Z 152,A -139.4626,B 17.5241,C -0.2907,E1 17.4067,E2 228.1397} C_DIS
LIN {X -97.1875,Y -82.6801,Z 152,A -141.0737,B 17.5241,C -0.29,E1 17.4037,E2 229.764} C_DIS
LIN {X -99.6184,Y -79.7353,Z 152,A -142.8113,B 17.5241,C -0.2932,E1 17.4007,E2 231.503} C_DIS
LIN {X -102.3749,Y -76.1629,Z 152,A -144.7061,B 17.5239,C -0.3021,E1 17.3975,E2 233.3812} C_DIS
LIN {X -103.9535,Y -73.9943,Z 152,A -145.9453,B 17.5239,C -0.3039,E1 17.3955,E2 234.6234} C_DIS
LIN {X -106.0012,Y -71.0296,Z 152,A -147.5443,B 17.5238,C -0.3084,E1 17.393,E2 236.2188} C_DIS
LIN {X -107.7088,Y -68.4131,Z 152,A -148.8533,B 17.5236,C -0.3149,E1 17.391,E2 237.516} C_DIS
LIN {X -109.2799,Y -65.8738,Z 152,A -150.3664,B 17.5236,C -0.3129,E1 17.3888,E2 239.0473} C_DIS
LIN {X -110.9285,Y -63.058,Z 152,A -151.8199,B 17.5236,C -0.317,E1 17.3868,E2 240.4982} C_DIS
LIN {X -112.3946,Y -60.4058,Z 152,A -153.222,B 17.5236,C -0.3193,E1 17.3849,E2 241.9037} C_DIS
Enddeposition()
END
